LIN {X 0,Y 340.799,Z 465.238,A -85,B 0,C 180,E1 -14193.019,E2 -14193.019} C_VEL
LIN {X 0,Y 340.748,Z 465.291,A -85,B 0,C 180,E1 -14195.638,E2 -14195.638} C_VEL
LIN {X 0,Y 340.726,Z 465.225,A -85,B 0,C 180,E1 -14199.473,E2 -14199.473} C_VEL
LIN {X 0,Y 340.851,Z 465.236,A -85,B 0,C 180,E1 -14201.984,E2 -14201.984} C_VEL
LIN {X 0,Y 340.863,Z 465.263,A -85,B 0,C 180,E1 -14205.705,E2 -14205.705} C_VEL
LIN {X 0,Y 340.864,Z 465.273,A -85,B 0,C 180,E1 -14209.306,E2 -14209.306} C_VEL
LIN {X 0,Y 341.054,Z 465.245,A -85,B 0,C 180,E1 -14212.898,E2 -14212.898} C_VEL
LIN {X 0,Y 341.162,Z 465.23,A -85,B 0,C 180,E1 -14217.638,E2 -14217.638} C_VEL
LIN {X 0,Y 341.269,Z 465.216,A -85,B 0,C 180,E1 -14220,E2 -14220} C_VEL
LIN {X 0,Y 341.163,Z 465.221,A -85,B 0,C 180,E1 -14222.361,E2 -14222.361} C_VEL
LIN {X 0,Y 341.054,Z 465.234,A -85,B 0,C 180,E1 -14227.102,E2 -14227.102} C_VEL
LIN {X 0,Y 340.863,Z 465.256,A -85,B 0,C 180,E1 -14230.694,E2 -14230.694} C_VEL
LIN {X 0,Y 340.856,Z 465.271,A -85,B 0,C 180,E1 -14234.325,E2 -14234.325} C_VEL
LIN {X 0,Y 340.83,Z 465.282,A -85,B 0,C 180,E1 -14238.466,E2 -14238.466} C_VEL
LIN {X 0,Y 340.713,Z 465.293,A -85,B 0,C 180,E1 -14241.843,E2 -14241.843} C_VEL
LIN {X 0,Y 340.764,Z 465.235,A -85,B 0,C 180,E1 -14245.665,E2 -14245.665} C_VEL
LIN {X 0,Y 340.735,Z 465.25,A -85,B 0,C 180,E1 -14248.32,E2 -14248.32} C_VEL
LIN {X 0,Y 340.697,Z 465.294,A -85,B 0,C 180,E1 -14251.044,E2 -14251.044} C_VEL
LIN {X 0,Y 340.712,Z 465.253,A -85,B 0,C 180,E1 -14255.279,E2 -14255.279} C_VEL
LIN {X 0,Y 340.719,Z 465.295,A -85,B 0,C 180,E1 -14258.39,E2 -14258.39} C_VEL
LIN {X 0,Y 340.719,Z 465.295,A -85,B 0,C 180,E1 -14261.304,E2 -14261.304} C_VEL
LIN {X 0,Y 340.717,Z 465.295,A -85,B 0,C 180,E1 -14264.532,E2 -14264.532} C_VEL
LIN {X 0,Y 340.728,Z 465.294,A -85,B 0,C 180,E1 -14267.948,E2 -14267.948} C_VEL
LIN {X 0,Y 340.723,Z 465.445,A -85,B 0,C 180,E1 -14269.848,E2 -14269.848} C_VEL
LIN {X 0,Y 341.012,Z 466.611,A -85,B 0,C 180,E1 -14270.401,E2 -14270.401} C_VEL
LIN {X 0,Y 342.25,Z 468.887,A -85,B 0,C 180,E1 -14271.014,E2 -14271.014} C_VEL
LIN {X 0,Y 344.629,Z 470.782,A -85,B 0,C 180,E1 -14272.06,E2 -14272.06} C_VEL
LIN {X 0,Y 345.88,Z 471.693,A -85,B 0,C 180,E1 -14272.605,E2 -14272.605} C_VEL
LIN {X 0,Y 347.625,Z 474.655,A -85,B 0,C 180,E1 -14273.477,E2 -14273.477} C_VEL
LIN {X 0,Y 350.309,Z 476.774,A -85,B 0,C 180,E1 -14274.708,E2 -14274.708} C_VEL
LIN {X 0,Y 351.421,Z 477.644,A -85,B 0,C 180,E1 -14275.211,E2 -14275.211} C_VEL
LIN {X 0,Y 353.186,Z 480.48,A -85,B 0,C 180,E1 -14276.141,E2 -14276.141} C_VEL
LIN {X 0,Y 355.66,Z 482.592,A -85,B 0,C 180,E1 -14277.346,E2 -14277.346} C_VEL
LIN {X 0,Y 357.075,Z 483.51,A -85,B 0,C 180,E1 -14278.024,E2 -14278.024} C_VEL
LIN {X 0,Y 359.092,Z 486.493,A -85,B 0,C 180,E1 -14279.137,E2 -14279.137} C_VEL
LIN {X 0,Y 361.635,Z 488.623,A -85,B 0,C 180,E1 -14280.474,E2 -14280.474} C_VEL
LIN {X 0,Y 363.122,Z 489.584,A -85,B 0,C 180,E1 -14281.247,E2 -14281.247} C_VEL
LIN {X 0,Y 365.429,Z 492.822,A -85,B 0,C 180,E1 -14282.618,E2 -14282.618} C_VEL
LIN {X 0,Y 368.413,Z 495.129,A -85,B 0,C 180,E1 -14284.366,E2 -14284.366} C_VEL
LIN {X 0,Y 369.281,Z 495.706,A -85,B 0,C 180,E1 -14284.883,E2 -14284.883} C_VEL
LIN {X 0,Y 371.456,Z 498.808,A -85,B 0,C 180,E1 -14286.343,E2 -14286.343} C_VEL
LIN {X 0,Y 373.823,Z 500.83,A -85,B 0,C 180,E1 -14287.914,E2 -14287.914} C_VEL
LIN {X 0,Y 375.91,Z 502.055,A -85,B 0,C 180,E1 -14289.347,E2 -14289.347} C_VEL
LIN {X 0,Y 377.976,Z 505.06,A -85,B 0,C 180,E1 -14291.017,E2 -14291.017} C_VEL
LIN {X 0,Y 380.522,Z 507.196,A -85,B 0,C 180,E1 -14293.159,E2 -14293.159} C_VEL
LIN {X 0,Y 382.957,Z 508.62,A -85,B 0,C 180,E1 -14295.383,E2 -14295.383} C_VEL
LIN {X 0,Y 384.39,Z 510.97,A -85,B 0,C 180,E1 -14297.071,E2 -14297.071} C_VEL
LIN {X 0,Y 386.194,Z 512.79,A -85,B 0,C 180,E1 -14299.323,E2 -14299.323} C_VEL
LIN {X 0,Y 387.761,Z 513.727,A -85,B 0,C 180,E1 -14301.663,E2 -14301.663} C_VEL
LIN {X 0,Y 389.276,Z 514.525,A -85,B 0,C 180,E1 -14304.821,E2 -14304.821} C_VEL
LIN {X 0,Y 389.886,Z 514.854,A -85,B 0,C 180,E1 -14306.9,E2 -14306.9} C_VEL
LIN {X 0,Y 390.177,Z 515.105,A -85,B 0,C 180,E1 -14308.968,E2 -14308.968} C_VEL
LIN {X 0,Y 390.177,Z 515.108,A -85,B 0,C 180,E1 -14311.032,E2 -14311.032} C_VEL
LIN {X 0,Y 389.886,Z 514.854,A -85,B 0,C 180,E1 -14313.1,E2 -14313.1} C_VEL
LIN {X 0,Y 389.276,Z 514.517,A -85,B 0,C 180,E1 -14315.179,E2 -14315.179} C_VEL
LIN {X 0,Y 388.018,Z 513.851,A -85,B 0,C 180,E1 -14317.882,E2 -14317.882} C_VEL
LIN {X 0,Y 386.325,Z 512.888,A -85,B 0,C 180,E1 -14320.481,E2 -14320.481} C_VEL
LIN {X 0,Y 384.529,Z 511.148,A -85,B 0,C 180,E1 -14322.765,E2 -14322.765} C_VEL
LIN {X 0,Y 383.033,Z 508.786,A -85,B 0,C 180,E1 -14324.521,E2 -14324.521} C_VEL
LIN {X 0,Y 381.452,Z 507.625,A -85,B 0,C 180,E1 -14326.043,E2 -14326.043} C_VEL
LIN {X 0,Y 378.941,Z 506.028,A -85,B 0,C 180,E1 -14328.17,E2 -14328.17} C_VEL
LIN {X 0,Y 376.883,Z 503.704,A -85,B 0,C 180,E1 -14329.842,E2 -14329.842} C_VEL
LIN {X 0,Y 375.682,Z 501.75,A -85,B 0,C 180,E1 -14330.82,E2 -14330.82} C_VEL
LIN {X 0,Y 372.73,Z 500.116,A -85,B 0,C 180,E1 -14332.801,E2 -14332.801} C_VEL
LIN {X 0,Y 370.289,Z 497.364,A -85,B 0,C 180,E1 -14334.444,E2 -14334.444} C_VEL
LIN {X 0,Y 368.921,Z 495.376,A -85,B 0,C 180,E1 -14335.338,E2 -14335.338} C_VEL
LIN {X 0,Y 365.831,Z 493.26,A -85,B 0,C 180,E1 -14337.137,E2 -14337.137} C_VEL
LIN {X 0,Y 363.334,Z 489.978,A -85,B 0,C 180,E1 -14338.618,E2 -14338.618} C_VEL
LIN {X 0,Y 362.471,Z 489.035,A -85,B 0,C 180,E1 -14339.107,E2 -14339.107} C_VEL
LIN {X 0,Y 359.635,Z 487.068,A -85,B 0,C 180,E1 -14340.582,E2 -14340.582} C_VEL
LIN {X 0,Y 357.4,Z 484.129,A -85,B 0,C 180,E1 -14341.799,E2 -14341.799} C_VEL
LIN {X 0,Y 356.762,Z 483.15,A -85,B 0,C 180,E1 -14342.132,E2 -14342.132} C_VEL
LIN {X 0,Y 353.946,Z 481.231,A -85,B 0,C 180,E1 -14343.494,E2 -14343.494} C_VEL
LIN {X 0,Y 351.935,Z 478.654,A -85,B 0,C 180,E1 -14344.511,E2 -14344.511} C_VEL
LIN {X 0,Y 351.246,Z 477.269,A -85,B 0,C 180,E1 -14344.88,E2 -14344.88} C_VEL
LIN {X 0,Y 348.17,Z 475.197,A -85,B 0,C 180,E1 -14346.279,E2 -14346.279} C_VEL
LIN {X 0,Y 346.328,Z 472.631,A -85,B 0,C 180,E1 -14347.157,E2 -14347.157} C_VEL
LIN {X 0,Y 345.416,Z 471.159,A -85,B 0,C 180,E1 -14347.617,E2 -14347.617} C_VEL
LIN {X 0,Y 342.655,Z 469.35,A -85,B 0,C 180,E1 -14348.796,E2 -14348.796} C_VEL
LIN {X 0,Y 341.302,Z 467.35,A -85,B 0,C 180,E1 -14349.427,E2 -14349.427} C_VEL
LIN {X 0,Y 340.805,Z 465.884,A -85,B 0,C 180,E1 -14349.863,E2 -14349.863} C_VEL
LIN {X 0,Y 340.725,Z 465.368,A -85,B 0,C 180,E1 -14350.255,E2 -14350.255} C_VEL
LIN {X 0,Y 340.701,Z 465.298,A -85,B 0,C 180,E1 -14353.782,E2 -14353.782} C_VEL
LIN {X 0,Y 340.734,Z 465.294,A -85,B 0,C 180,E1 -14357.105,E2 -14357.105} C_VEL
LIN {X 0,Y 340.73,Z 465.294,A -85,B 0,C 180,E1 -14360.252,E2 -14360.252} C_VEL
LIN {X 0,Y 340.706,Z 465.281,A -85,B 0,C 180,E1 -14363.558,E2 -14363.558} C_VEL
LIN {X 0,Y 340.685,Z 465.246,A -85,B 0,C 180,E1 -14366.153,E2 -14366.153} C_VEL
LIN {X 0,Y 340.768,Z 465.28,A -85,B 0,C 180,E1 -14370.332,E2 -14370.332} C_VEL
LIN {X 0,Y 340.797,Z 465.225,A -85,B 0,C 180,E1 -14373.02,E2 -14373.02} C_VEL
LIN {X 0,Y 340.752,Z 465.241,A -85,B 0,C 180,E1 -14374.696,E2 -14374.696} C_VEL
LIN {X 0,Y 340.069,Z 465.349,A -85,B 0,C 180,E1 -14375.682,E2 -14375.682} C_VEL
LIN {X 0,Y 337.172,Z 465.738,A -85,B 0,C 180,E1 -14377.286,E2 -14377.286} C_VEL
LIN {X 0,Y 334.749,Z 466.031,A -85,B 0,C 180,E1 -14378.585,E2 -14378.585} C_VEL
LIN {X 0,Y 333.75,Z 466.146,A -85,B 0,C 180,E1 -14379.592,E2 -14379.592} C_VEL
LIN {X 0,Y 333.69,Z 466.154,A -85,B 0,C 180,E1 -14379.932,E2 -14379.932} C_VEL
LIN {X 0,Y 333.738,Z 466.154,A -85,B 0,C 180,E1 -14382.854,E2 -14382.854} C_VEL
LIN {X 0,Y 333.789,Z 466.155,A -85,B 0,C 180,E1 -14386.609,E2 -14386.609} C_VEL
LIN {X 0,Y 333.853,Z 466.142,A -85,B 0,C 180,E1 -14390.305,E2 -14390.305} C_VEL
LIN {X 0,Y 334.006,Z 466.114,A -85,B 0,C 180,E1 -14392.747,E2 -14392.747} C_VEL
LIN {X 0,Y 333.805,Z 466.147,A -85,B 0,C 180,E1 -14395.169,E2 -14395.169} C_VEL
LIN {X 0,Y 334.1,Z 466.103,A -85,B 0,C 180,E1 -14397.589,E2 -14397.589} C_VEL
LIN {X 0,Y 334.221,Z 466.094,A -85,B 0,C 180,E1 -14400,E2 -14400} C_VEL
LIN {X 0,Y 334.099,Z 466.109,A -85,B 0,C 180,E1 -14402.411,E2 -14402.411} C_VEL
LIN {X 0,Y 334.01,Z 466.129,A -85,B 0,C 180,E1 -14406.039,E2 -14406.039} C_VEL
LIN {X 0,Y 333.952,Z 466.115,A -85,B 0,C 180,E1 -14408.472,E2 -14408.472} C_VEL
LIN {X 0,Y 333.784,Z 466.146,A -85,B 0,C 180,E1 -14412.155,E2 -14412.155} C_VEL
LIN {X 0,Y 333.771,Z 466.158,A -85,B 0,C 180,E1 -14415.887,E2 -14415.887} C_VEL
LIN {X 0,Y 333.789,Z 466.1,A -85,B 0,C 180,E1 -14418.655,E2 -14418.655} C_VEL
LIN {X 0,Y 333.65,Z 466.134,A -85,B 0,C 180,E1 -14422.281,E2 -14422.281} C_VEL
LIN {X 0,Y 333.73,Z 466.133,A -85,B 0,C 180,E1 -14426.247,E2 -14426.247} C_VEL
LIN {X 0,Y 333.706,Z 466.111,A -85,B 0,C 180,E1 -14428.973,E2 -14428.973} C_VEL
LIN {X 0,Y 333.646,Z 466.172,A -85,B 0,C 180,E1 -14432.59,E2 -14432.59} C_VEL
LIN {X 0,Y 333.672,Z 466.144,A -85,B 0,C 180,E1 -14436.139,E2 -14436.139} C_VEL
LIN {X 0,Y 333.678,Z 466.146,A -85,B 0,C 180,E1 -14439.188,E2 -14439.188} C_VEL
LIN {X 0,Y 333.708,Z 466.29,A -85,B 0,C 180,E1 -14441.258,E2 -14441.258} C_VEL
LIN {X 0,Y 336.781,Z 476.03,A -85,B 0,C 180,E1 -14444.671,E2 -14444.671} C_VEL
LIN {X 0,Y 337.849,Z 478.396,A -85,B 0,C 180,E1 -14445.014,E2 -14445.014} C_VEL
LIN {X 0,Y 341.276,Z 483.882,A -85,B 0,C 180,E1 -14445.739,E2 -14445.739} C_VEL
LIN {X 0,Y 349.072,Z 497.083,A -85,B 0,C 180,E1 -14447.326,E2 -14447.326} C_VEL
LIN {X 0,Y 358.673,Z 515.254,A -85,B 0,C 180,E1 -14449.186,E2 -14449.186} C_VEL
LIN {X 0,Y 366.818,Z 532.432,A -85,B 0,C 180,E1 -14450.694,E2 -14450.694} C_VEL
LIN {X 0,Y 368.049,Z 538.307,A -85,B 0,C 180,E1 -14450.994,E2 -14450.994} C_VEL
LIN {X 0,Y 363.639,Z 661.533,A -85,B 0,C 180,E1 -14453.452,E2 -14453.452} C_VEL
LIN {X 0,Y 362.413,Z 691.653,A -85,B 0,C 180,E1 -14454.084,E2 -14454.084} C_VEL
LIN {X 0,Y 361.365,Z 705.109,A -85,B 0,C 180,E1 -14454.479,E2 -14454.479} C_VEL
LIN {X 0,Y 359.961,Z 718.486,A -85,B 0,C 180,E1 -14455.005,E2 -14455.005} C_VEL
LIN {X 0,Y 358.069,Z 734.159,A -85,B 0,C 180,E1 -14455.818,E2 -14455.818} C_VEL
LIN {X 0,Y 355.544,Z 750.452,A -85,B 0,C 180,E1 -14456.904,E2 -14456.904} C_VEL
LIN {X 0,Y 353.23,Z 763.836,A -85,B 0,C 180,E1 -14458.013,E2 -14458.013} C_VEL
LIN {X 0,Y 350.74,Z 776.671,A -85,B 0,C 180,E1 -14459.274,E2 -14459.274} C_VEL
LIN {X 0,Y 348.622,Z 786.926,A -85,B 0,C 180,E1 -14460.442,E2 -14460.442} C_VEL
LIN {X 0,Y 346.254,Z 797.637,A -85,B 0,C 180,E1 -14461.842,E2 -14461.842} C_VEL
LIN {X 0,Y 344.049,Z 807.328,A -85,B 0,C 180,E1 -14463.295,E2 -14463.295} C_VEL
LIN {X 0,Y 342.031,Z 816.281,A -85,B 0,C 180,E1 -14464.827,E2 -14464.827} C_VEL
LIN {X 0,Y 339.631,Z 826.499,A -85,B 0,C 180,E1 -14466.849,E2 -14466.849} C_VEL
LIN {X 0,Y 337.855,Z 834.392,A -85,B 0,C 180,E1 -14468.653,E2 -14468.653} C_VEL
LIN {X 0,Y 336.381,Z 841.359,A -85,B 0,C 180,E1 -14470.471,E2 -14470.471} C_VEL
LIN {X 0,Y 335.184,Z 847.502,A -85,B 0,C 180,E1 -14472.301,E2 -14472.301} C_VEL
LIN {X 0,Y 333.91,Z 854.451,A -85,B 0,C 180,E1 -14474.747,E2 -14474.747} C_VEL
LIN {X 0,Y 332.975,Z 860.207,A -85,B 0,C 180,E1 -14477.196,E2 -14477.196} C_VEL
LIN {X 0,Y 332.45,Z 863.818,A -85,B 0,C 180,E1 -14479.032,E2 -14479.032} C_VEL
LIN {X 0,Y 332.118,Z 867.67,A -85,B 0,C 180,E1 -14481.482,E2 -14481.482} C_VEL
LIN {X 0,Y 332.029,Z 870.521,A -85,B 0,C 180,E1 -14483.925,E2 -14483.925} C_VEL
LIN {X 0,Y 331.964,Z 872.403,A -85,B 0,C 180,E1 -14486.359,E2 -14486.359} C_VEL
LIN {X 0,Y 331.902,Z 873.076,A -85,B 0,C 180,E1 -14487.573,E2 -14487.573} C_VEL
LIN {X 0,Y 331.911,Z 873.548,A -85,B 0,C 180,E1 -14490,E2 -14490} C_VEL
LIN {X 0,Y 331.902,Z 873.076,A -85,B 0,C 180,E1 -14492.427,E2 -14492.427} C_VEL
LIN {X 0,Y 331.936,Z 871.654,A -85,B 0,C 180,E1 -14494.858,E2 -14494.858} C_VEL
LIN {X 0,Y 332.033,Z 869.271,A -85,B 0,C 180,E1 -14497.296,E2 -14497.296} C_VEL
LIN {X 0,Y 332.347,Z 864.858,A -85,B 0,C 180,E1 -14500.355,E2 -14500.355} C_VEL
LIN {X 0,Y 332.783,Z 861.493,A -85,B 0,C 180,E1 -14502.192,E2 -14502.192} C_VEL
LIN {X 0,Y 333.616,Z 855.994,A -85,B 0,C 180,E1 -14504.643,E2 -14504.643} C_VEL
LIN {X 0,Y 334.458,Z 851.135,A -85,B 0,C 180,E1 -14506.479,E2 -14506.479} C_VEL
LIN {X 0,Y 335.999,Z 843.467,A -85,B 0,C 180,E1 -14508.917,E2 -14508.917} C_VEL
LIN {X 0,Y 337.306,Z 836.81,A -85,B 0,C 180,E1 -14510.744,E2 -14510.744} C_VEL
LIN {X 0,Y 339.006,Z 829.257,A -85,B 0,C 180,E1 -14512.552,E2 -14512.552} C_VEL
LIN {X 0,Y 341.098,Z 820.675,A -85,B 0,C 180,E1 -14514.335,E2 -14514.335} C_VEL
LIN {X 0,Y 343.221,Z 810.88,A -85,B 0,C 180,E1 -14516.119,E2 -14516.119} C_VEL
LIN {X 0,Y 345.731,Z 799.648,A -85,B 0,C 180,E1 -14517.874,E2 -14517.874} C_VEL
LIN {X 0,Y 348.088,Z 789.167,A -85,B 0,C 180,E1 -14519.282,E2 -14519.282} C_VEL
LIN {X 0,Y 350.131,Z 779.54,A -85,B 0,C 180,E1 -14520.419,E2 -14520.419} C_VEL
LIN {X 0,Y 352.331,Z 768.335,A -85,B 0,C 180,E1 -14521.574,E2 -14521.574} C_VEL
LIN {X 0,Y 354.632,Z 755.677,A -85,B 0,C 180,E1 -14522.685,E2 -14522.685} C_VEL
LIN {X 0,Y 356.641,Z 743.661,A -85,B 0,C 180,E1 -14523.572,E2 -14523.572} C_VEL
LIN {X 0,Y 358.505,Z 730.453,A -85,B 0,C 180,E1 -14524.39,E2 -14524.39} C_VEL
LIN {X 0,Y 360.135,Z 717.326,A -85,B 0,C 180,E1 -14525.04,E2 -14525.04} C_VEL
LIN {X 0,Y 361.468,Z 704.407,A -85,B 0,C 180,E1 -14525.54,E2 -14525.54} C_VEL
LIN {X 0,Y 362.415,Z 691.653,A -85,B 0,C 180,E1 -14525.916,E2 -14525.916} C_VEL
LIN {X 0,Y 363.878,Z 654.368,A -85,B 0,C 180,E1 -14526.692,E2 -14526.692} C_VEL
LIN {X 0,Y 367.077,Z 565.249,A -85,B 0,C 180,E1 -14528.468,E2 -14528.468} C_VEL
LIN {X 0,Y 368.055,Z 538.146,A -85,B 0,C 180,E1 -14529.01,E2 -14529.01} C_VEL
LIN {X 0,Y 366.541,Z 531.775,A -85,B 0,C 180,E1 -14529.358,E2 -14529.358} C_VEL
LIN {X 0,Y 357.488,Z 512.916,A -85,B 0,C 180,E1 -14531.038,E2 -14531.038} C_VEL
LIN {X 0,Y 348.525,Z 496.099,A -85,B 0,C 180,E1 -14532.783,E2 -14532.783} C_VEL
LIN {X 0,Y 339.359,Z 480.633,A -85,B 0,C 180,E1 -14534.669,E2 -14534.669} C_VEL
LIN {X 0,Y 336.838,Z 476.211,A -85,B 0,C 180,E1 -14535.284,E2 -14535.284} C_VEL
LIN {X 0,Y 333.701,Z 466.326,A -85,B 0,C 180,E1 -14538.741,E2 -14538.741} C_VEL
LIN {X 0,Y 333.651,Z 466.176,A -85,B 0,C 180,E1 -14542.349,E2 -14542.349} C_VEL
LIN {X 0,Y 333.669,Z 466.135,A -85,B 0,C 180,E1 -14545.341,E2 -14545.341} C_VEL
LIN {X 0,Y 333.639,Z 466.176,A -85,B 0,C 180,E1 -14548.223,E2 -14548.223} C_VEL
LIN {X 0,Y 333.706,Z 466.111,A -85,B 0,C 180,E1 -14551.027,E2 -14551.027} C_VEL
LIN {X 0,Y 333.73,Z 466.132,A -85,B 0,C 180,E1 -14553.753,E2 -14553.753} C_VEL
LIN {X 0,Y 333.65,Z 466.134,A -85,B 0,C 180,E1 -14557.719,E2 -14557.719} C_VEL
LIN {X 0,Y 333.787,Z 466.104,A -85,B 0,C 180,E1 -14561.589,E2 -14561.589} C_VEL
LIN {X 0,Y 333.802,Z 466.143,A -85,B 0,C 180,E1 -14565.576,E2 -14565.576} C_VEL
LIN {X 0,Y 333.827,Z 466.15,A -85,B 0,C 180,E1 -14569.078,E2 -14569.078} C_VEL
LIN {X 0,Y 334.001,Z 466.121,A -85,B 0,C 180,E1 -14572.747,E2 -14572.747} C_VEL
LIN {X 0,Y 333.805,Z 466.146,A -85,B 0,C 180,E1 -14575.169,E2 -14575.169} C_VEL
LIN {X 0,Y 334.1,Z 466.108,A -85,B 0,C 180,E1 -14577.589,E2 -14577.589} C_VEL
LIN {X 0,Y 334.221,Z 466.093,A -85,B 0,C 180,E1 -14580,E2 -14580} C_VEL
LIN {X 0,Y 334.1,Z 466.1,A -85,B 0,C 180,E1 -14582.411,E2 -14582.411} C_VEL
LIN {X 0,Y 333.989,Z 466.11,A -85,B 0,C 180,E1 -14586.616,E2 -14586.616} C_VEL
LIN {X 0,Y 333.853,Z 466.141,A -85,B 0,C 180,E1 -14589.695,E2 -14589.695} C_VEL
LIN {X 0,Y 333.789,Z 466.155,A -85,B 0,C 180,E1 -14593.391,E2 -14593.391} C_VEL
LIN {X 0,Y 333.738,Z 466.154,A -85,B 0,C 180,E1 -14597.146,E2 -14597.146} C_VEL
LIN {X 0,Y 333.725,Z 466.152,A -85,B 0,C 180,E1 -14599.691,E2 -14599.691} C_VEL
LIN {X 0,Y 333.664,Z 466.164,A -85,B 0,C 180,E1 -14603.59,E2 -14603.59} C_VEL
LIN {X 0,Y 333.728,Z 466.104,A -85,B 0,C 180,E1 -14606.246,E2 -14606.246} C_VEL
LIN {X 0,Y 333.704,Z 466.14,A -85,B 0,C 180,E1 -14608.972,E2 -14608.972} C_VEL
LIN {X 0,Y 333.636,Z 466.136,A -85,B 0,C 180,E1 -14612.587,E2 -14612.587} C_VEL
LIN {X 0,Y 333.671,Z 466.147,A -85,B 0,C 180,E1 -14616.139,E2 -14616.139} C_VEL
LIN {X 0,Y 333.681,Z 466.173,A -85,B 0,C 180,E1 -14619.187,E2 -14619.187} C_VEL
LIN {X 0,Y 333.683,Z 466.171,A -85,B 0,C 180,E1 -14622.511,E2 -14622.511} C_VEL
LIN {X 0,Y 333.653,Z 466.174,A -85,B 0,C 180,E1 -14625.966,E2 -14625.966} C_VEL
LIN {X 0,Y 333.716,Z 466.35,A -85,B 0,C 180,E1 -14627.284,E2 -14627.284} C_VEL
LIN {X 0,Y 334.001,Z 467.585,A -85,B 0,C 180,E1 -14627.8,E2 -14627.8} C_VEL
LIN {X 0,Y 335.396,Z 469.981,A -85,B 0,C 180,E1 -14628.466,E2 -14628.466} C_VEL
LIN {X 0,Y 337.884,Z 471.863,A -85,B 0,C 180,E1 -14629.485,E2 -14629.485} C_VEL
LIN {X 0,Y 338.798,Z 472.664,A -85,B 0,C 180,E1 -14629.887,E2 -14629.887} C_VEL
LIN {X 0,Y 340.366,Z 475.312,A -85,B 0,C 180,E1 -14630.625,E2 -14630.625} C_VEL
LIN {X 0,Y 342.872,Z 477.456,A -85,B 0,C 180,E1 -14631.722,E2 -14631.722} C_VEL
LIN {X 0,Y 344.061,Z 478.298,A -85,B 0,C 180,E1 -14632.229,E2 -14632.229} C_VEL
LIN {X 0,Y 346.074,Z 481.409,A -85,B 0,C 180,E1 -14633.214,E2 -14633.214} C_VEL
LIN {X 0,Y 348.838,Z 483.58,A -85,B 0,C 180,E1 -14634.467,E2 -14634.467} C_VEL
LIN {X 0,Y 349.69,Z 484.296,A -85,B 0,C 180,E1 -14634.863,E2 -14634.863} C_VEL
LIN {X 0,Y 351.781,Z 487.31,A -85,B 0,C 180,E1 -14635.92,E2 -14635.92} C_VEL
LIN {X 0,Y 354.617,Z 489.628,A -85,B 0,C 180,E1 -14637.289,E2 -14637.289} C_VEL
LIN {X 0,Y 355.598,Z 490.455,A -85,B 0,C 180,E1 -14637.775,E2 -14637.775} C_VEL
LIN {X 0,Y 358.077,Z 493.716,A -85,B 0,C 180,E1 -14639.102,E2 -14639.102} C_VEL
LIN {X 0,Y 360.763,Z 495.744,A -85,B 0,C 180,E1 -14640.497,E2 -14640.497} C_VEL
LIN {X 0,Y 361.761,Z 496.461,A -85,B 0,C 180,E1 -14641.011,E2 -14641.011} C_VEL
LIN {X 0,Y 364.25,Z 499.79,A -85,B 0,C 180,E1 -14642.469,E2 -14642.469} C_VEL
LIN {X 0,Y 367.384,Z 502.135,A -85,B 0,C 180,E1 -14644.289,E2 -14644.289} C_VEL
LIN {X 0,Y 368.211,Z 502.958,A -85,B 0,C 180,E1 -14644.805,E2 -14644.805} C_VEL
LIN {X 0,Y 370.641,Z 506.172,A -85,B 0,C 180,E1 -14646.411,E2 -14646.411} C_VEL
LIN {X 0,Y 373.648,Z 508.333,A -85,B 0,C 180,E1 -14648.402,E2 -14648.402} C_VEL
LIN {X 0,Y 374.774,Z 509.041,A -85,B 0,C 180,E1 -14649.188,E2 -14649.188} C_VEL
LIN {X 0,Y 376.863,Z 511.983,A -85,B 0,C 180,E1 -14650.848,E2 -14650.848} C_VEL
LIN {X 0,Y 379.588,Z 514.233,A -85,B 0,C 180,E1 -14653.116,E2 -14653.116} C_VEL
LIN {X 0,Y 381.909,Z 515.568,A -85,B 0,C 180,E1 -14655.207,E2 -14655.207} C_VEL
LIN {X 0,Y 383.479,Z 518.067,A -85,B 0,C 180,E1 -14657.039,E2 -14657.039} C_VEL
LIN {X 0,Y 385.431,Z 519.973,A -85,B 0,C 180,E1 -14659.494,E2 -14659.494} C_VEL
LIN {X 0,Y 387.14,Z 520.894,A -85,B 0,C 180,E1 -14662.101,E2 -14662.101} C_VEL
LIN {X 0,Y 388.408,Z 521.561,A -85,B 0,C 180,E1 -14664.809,E2 -14664.809} C_VEL
LIN {X 0,Y 389.019,Z 521.9,A -85,B 0,C 180,E1 -14666.893,E2 -14666.893} C_VEL
LIN {X 0,Y 389.312,Z 522.151,A -85,B 0,C 180,E1 -14668.966,E2 -14668.966} C_VEL
LIN {X 0,Y 389.312,Z 522.154,A -85,B 0,C 180,E1 -14671.034,E2 -14671.034} C_VEL
LIN {X 0,Y 389.019,Z 521.9,A -85,B 0,C 180,E1 -14673.107,E2 -14673.107} C_VEL
LIN {X 0,Y 388.31,Z 521.48,A -85,B 0,C 180,E1 -14675.48,E2 -14675.48} C_VEL
LIN {X 0,Y 386.879,Z 520.77,A -85,B 0,C 180,E1 -14678.356,E2 -14678.356} C_VEL
LIN {X 0,Y 385.035,Z 519.643,A -85,B 0,C 180,E1 -14681.047,E2 -14681.047} C_VEL
LIN {X 0,Y 383.292,Z 517.821,A -85,B 0,C 180,E1 -14683.19,E2 -14683.19} C_VEL
LIN {X 0,Y 381.547,Z 515.224,A -85,B 0,C 180,E1 -14685.156,E2 -14685.156} C_VEL
LIN {X 0,Y 378.664,Z 513.605,A -85,B 0,C 180,E1 -14687.681,E2 -14687.681} C_VEL
LIN {X 0,Y 376.317,Z 511.354,A -85,B 0,C 180,E1 -14689.572,E2 -14689.572} C_VEL
LIN {X 0,Y 374.469,Z 508.696,A -85,B 0,C 180,E1 -14691.032,E2 -14691.032} C_VEL
LIN {X 0,Y 371.535,Z 506.981,A -85,B 0,C 180,E1 -14693.005,E2 -14693.005} C_VEL
LIN {X 0,Y 368.963,Z 504.114,A -85,B 0,C 180,E1 -14694.717,E2 -14694.717} C_VEL
LIN {X 0,Y 367.639,Z 502.248,A -85,B 0,C 180,E1 -14695.563,E2 -14695.563} C_VEL
LIN {X 0,Y 364.568,Z 500.105,A -85,B 0,C 180,E1 -14697.345,E2 -14697.345} C_VEL
LIN {X 0,Y 361.995,Z 496.856,A -85,B 0,C 180,E1 -14698.851,E2 -14698.851} C_VEL
LIN {X 0,Y 361.33,Z 496.008,A -85,B 0,C 180,E1 -14699.218,E2 -14699.218} C_VEL
LIN {X 0,Y 358.483,Z 494.098,A -85,B 0,C 180,E1 -14700.689,E2 -14700.689} C_VEL
LIN {X 0,Y 355.928,Z 490.993,A -85,B 0,C 180,E1 -14702.049,E2 -14702.049} C_VEL
LIN {X 0,Y 355.336,Z 489.998,A -85,B 0,C 180,E1 -14702.366,E2 -14702.366} C_VEL
LIN {X 0,Y 352.412,Z 487.954,A -85,B 0,C 180,E1 -14703.77,E2 -14703.77} C_VEL
LIN {X 0,Y 350.116,Z 485.046,A -85,B 0,C 180,E1 -14704.922,E2 -14704.922} C_VEL
LIN {X 0,Y 349.317,Z 483.857,A -85,B 0,C 180,E1 -14705.316,E2 -14705.316} C_VEL
LIN {X 0,Y 346.252,Z 481.607,A -85,B 0,C 180,E1 -14706.704,E2 -14706.704} C_VEL
LIN {X 0,Y 344.287,Z 478.716,A -85,B 0,C 180,E1 -14707.664,E2 -14707.664} C_VEL
LIN {X 0,Y 343.675,Z 477.863,A -85,B 0,C 180,E1 -14707.943,E2 -14707.943} C_VEL
LIN {X 0,Y 340.917,Z 475.912,A -85,B 0,C 180,E1 -14709.138,E2 -14709.138} C_VEL
LIN {X 0,Y 339.142,Z 473.436,A -85,B 0,C 180,E1 -14709.938,E2 -14709.938} C_VEL
LIN {X 0,Y 338.385,Z 472.108,A -85,B 0,C 180,E1 -14710.305,E2 -14710.305} C_VEL
LIN {X 0,Y 335.698,Z 470.334,A -85,B 0,C 180,E1 -14711.401,E2 -14711.401} C_VEL
LIN {X 0,Y 334.143,Z 467.942,A -85,B 0,C 180,E1 -14712.123,E2 -14712.123} C_VEL
LIN {X 0,Y 333.767,Z 466.637,A -85,B 0,C 180,E1 -14712.526,E2 -14712.526} C_VEL
LIN {X 0,Y 333.668,Z 466.18,A -85,B 0,C 180,E1 -14713.215,E2 -14713.215} C_VEL
LIN {X 0,Y 333.663,Z 466.174,A -85,B 0,C 180,E1 -14715.967,E2 -14715.967} C_VEL
LIN {X 0,Y 333.695,Z 466.17,A -85,B 0,C 180,E1 -14719.304,E2 -14719.304} C_VEL
LIN {X 0,Y 333.662,Z 466.169,A -85,B 0,C 180,E1 -14723.167,E2 -14723.167} C_VEL
LIN {X 0,Y 333.667,Z 466.122,A -85,B 0,C 180,E1 -14725.341,E2 -14725.341} C_VEL
LIN {X 0,Y 333.696,Z 466.169,A -85,B 0,C 180,E1 -14729.71,E2 -14729.71} C_VEL
LIN {X 0,Y 333.737,Z 466.108,A -85,B 0,C 180,E1 -14732.401,E2 -14732.401} C_VEL
LIN {X 0,Y 333.718,Z 466.124,A -85,B 0,C 180,E1 -14735.09,E2 -14735.09} C_VEL
LIN {X 0,Y 333.666,Z 466.158,A -85,B 0,C 180,E1 -14739.019,E2 -14739.019} C_VEL
LIN {X 0,Y 333.69,Z 466.154,A -85,B 0,C 180,E1 -14739.932,E2 -14739.932} C_VEL
LIN {X 0,Y 333.082,Z 466.24,A -85,B 0,C 180,E1 -14740.939,E2 -14740.939} C_VEL
LIN {X 0,Y 330.26,Z 466.592,A -85,B 0,C 180,E1 -14742.579,E2 -14742.579} C_VEL
LIN {X 0,Y 327.845,Z 466.883,A -85,B 0,C 180,E1 -14743.907,E2 -14743.907} C_VEL
LIN {X 0,Y 326.824,Z 467.008,A -85,B 0,C 180,E1 -14744.935,E2 -14744.935} C_VEL
LIN {X 0,Y 326.75,Z 467.021,A -85,B 0,C 180,E1 -14745.283,E2 -14745.283} C_VEL
LIN {X 0,Y 326.762,Z 467.011,A -85,B 0,C 180,E1 -14748.839,E2 -14748.839} C_VEL
LIN {X 0,Y 326.96,Z 466.993,A -85,B 0,C 180,E1 -14752.59,E2 -14752.59} C_VEL
LIN {X 0,Y 326.772,Z 467.022,A -85,B 0,C 180,E1 -14755.065,E2 -14755.065} C_VEL
LIN {X 0,Y 327.041,Z 466.982,A -85,B 0,C 180,E1 -14757.537,E2 -14757.537} C_VEL
LIN {X 0,Y 327.173,Z 466.972,A -85,B 0,C 180,E1 -14760,E2 -14760} C_VEL
LIN {X 0,Y 327.04,Z 466.987,A -85,B 0,C 180,E1 -14762.464,E2 -14762.464} C_VEL
LIN {X 0,Y 326.985,Z 467.003,A -85,B 0,C 180,E1 -14766.17,E2 -14766.17} C_VEL
LIN {X 0,Y 326.799,Z 467.016,A -85,B 0,C 180,E1 -14769.907,E2 -14769.907} C_VEL
LIN {X 0,Y 326.752,Z 467.014,A -85,B 0,C 180,E1 -14773.686,E2 -14773.686} C_VEL
LIN {X 0,Y 326.692,Z 467.01,A -85,B 0,C 180,E1 -14777.528,E2 -14777.528} C_VEL
LIN {X 0,Y 326.651,Z 466.974,A -85,B 0,C 180,E1 -14780.136,E2 -14780.136} C_VEL
LIN {X 0,Y 326.643,Z 467.048,A -85,B 0,C 180,E1 -14784.13,E2 -14784.13} C_VEL
LIN {X 0,Y 326.679,Z 466.995,A -85,B 0,C 180,E1 -14786.858,E2 -14786.858} C_VEL
LIN {X 0,Y 326.636,Z 467.02,A -85,B 0,C 180,E1 -14790.613,E2 -14790.613} C_VEL
LIN {X 0,Y 326.604,Z 467.019,A -85,B 0,C 180,E1 -14794.02,E2 -14794.02} C_VEL
LIN {X 0,Y 326.625,Z 467.045,A -85,B 0,C 180,E1 -14797.24,E2 -14797.24} C_VEL
LIN {X 0,Y 326.65,Z 467.151,A -85,B 0,C 180,E1 -14800.2,E2 -14800.2} C_VEL
LIN {X 0,Y 329.467,Z 475.897,A -85,B 0,C 180,E1 -14803.415,E2 -14803.415} C_VEL
LIN {X 0,Y 332.332,Z 480.715,A -85,B 0,C 180,E1 -14804.132,E2 -14804.132} C_VEL
LIN {X 0,Y 339.589,Z 492.764,A -85,B 0,C 180,E1 -14805.72,E2 -14805.72} C_VEL
LIN {X 0,Y 347.23,Z 506.263,A -85,B 0,C 180,E1 -14807.3,E2 -14807.3} C_VEL
LIN {X 0,Y 356.44,Z 524.382,A -85,B 0,C 180,E1 -14809.115,E2 -14809.115} C_VEL
LIN {X 0,Y 361.7,Z 535.896,A -85,B 0,C 180,E1 -14810.119,E2 -14810.119} C_VEL
LIN {X 0,Y 362.496,Z 539.647,A -85,B 0,C 180,E1 -14810.318,E2 -14810.318} C_VEL
LIN {X 0,Y 357.961,Z 661.323,A -85,B 0,C 180,E1 -14812.775,E2 -14812.775} C_VEL
LIN {X 0,Y 356.676,Z 691.443,A -85,B 0,C 180,E1 -14813.413,E2 -14813.413} C_VEL
LIN {X 0,Y 355.524,Z 705.9,A -85,B 0,C 180,E1 -14813.848,E2 -14813.848} C_VEL
LIN {X 0,Y 353.84,Z 721.343,A -85,B 0,C 180,E1 -14814.483,E2 -14814.483} C_VEL
LIN {X 0,Y 351.496,Z 738.469,A -85,B 0,C 180,E1 -14815.448,E2 -14815.448} C_VEL
LIN {X 0,Y 349.258,Z 751.982,A -85,B 0,C 180,E1 -14816.402,E2 -14816.402} C_VEL
LIN {X 0,Y 347.187,Z 763.625,A -85,B 0,C 180,E1 -14817.388,E2 -14817.388} C_VEL
LIN {X 0,Y 344.58,Z 776.454,A -85,B 0,C 180,E1 -14818.662,E2 -14818.662} C_VEL
LIN {X 0,Y 342.294,Z 787.09,A -85,B 0,C 180,E1 -14819.896,E2 -14819.896} C_VEL
LIN {X 0,Y 339.677,Z 798.43,A -85,B 0,C 180,E1 -14821.416,E2 -14821.416} C_VEL
LIN {X 0,Y 337.178,Z 808.891,A -85,B 0,C 180,E1 -14823.042,E2 -14823.042} C_VEL
LIN {X 0,Y 335.326,Z 816.805,A -85,B 0,C 180,E1 -14824.444,E2 -14824.444} C_VEL
LIN {X 0,Y 333.006,Z 826.285,A -85,B 0,C 180,E1 -14826.361,E2 -14826.361} C_VEL
LIN {X 0,Y 331.131,Z 834.179,A -85,B 0,C 180,E1 -14828.197,E2 -14828.197} C_VEL
LIN {X 0,Y 329.332,Z 842.198,A -85,B 0,C 180,E1 -14830.361,E2 -14830.361} C_VEL
LIN {X 0,Y 327.907,Z 849.105,A -85,B 0,C 180,E1 -14832.539,E2 -14832.539} C_VEL
LIN {X 0,Y 326.94,Z 854.237,A -85,B 0,C 180,E1 -14834.413,E2 -14834.413} C_VEL
LIN {X 0,Y 326.222,Z 858.709,A -85,B 0,C 180,E1 -14836.292,E2 -14836.292} C_VEL
LIN {X 0,Y 325.427,Z 863.607,A -85,B 0,C 180,E1 -14838.793,E2 -14838.793} C_VEL
LIN {X 0,Y 325.047,Z 867.458,A -85,B 0,C 180,E1 -14841.295,E2 -14841.295} C_VEL
LIN {X 0,Y 324.944,Z 870.311,A -85,B 0,C 180,E1 -14843.792,E2 -14843.792} C_VEL
LIN {X 0,Y 324.869,Z 872.193,A -85,B 0,C 180,E1 -14846.279,E2 -14846.279} C_VEL
LIN {X 0,Y 324.822,Z 872.867,A -85,B 0,C 180,E1 -14847.52,E2 -14847.52} C_VEL
LIN {X 0,Y 324.818,Z 873.339,A -85,B 0,C 180,E1 -14850,E2 -14850} C_VEL
LIN {X 0,Y 324.822,Z 872.867,A -85,B 0,C 180,E1 -14852.48,E2 -14852.48} C_VEL
LIN {X 0,Y 324.85,Z 871.444,A -85,B 0,C 180,E1 -14854.964,E2 -14854.964} C_VEL
LIN {X 0,Y 324.948,Z 869.06,A -85,B 0,C 180,E1 -14857.456,E2 -14857.456} C_VEL
LIN {X 0,Y 325.283,Z 864.646,A -85,B 0,C 180,E1 -14860.582,E2 -14860.582} C_VEL
LIN {X 0,Y 325.747,Z 861.28,A -85,B 0,C 180,E1 -14862.459,E2 -14862.459} C_VEL
LIN {X 0,Y 326.667,Z 855.782,A -85,B 0,C 180,E1 -14864.961,E2 -14864.961} C_VEL
LIN {X 0,Y 327.566,Z 850.922,A -85,B 0,C 180,E1 -14866.836,E2 -14866.836} C_VEL
LIN {X 0,Y 329.157,Z 843.253,A -85,B 0,C 180,E1 -14869.326,E2 -14869.326} C_VEL
LIN {X 0,Y 330.56,Z 836.597,A -85,B 0,C 180,E1 -14871.188,E2 -14871.188} C_VEL
LIN {X 0,Y 332.334,Z 829.043,A -85,B 0,C 180,E1 -14873.03,E2 -14873.03} C_VEL
LIN {X 0,Y 334.53,Z 820.462,A -85,B 0,C 180,E1 -14874.845,E2 -14874.845} C_VEL
LIN {X 0,Y 336.776,Z 810.667,A -85,B 0,C 180,E1 -14876.658,E2 -14876.658} C_VEL
LIN {X 0,Y 339.154,Z 800.442,A -85,B 0,C 180,E1 -14878.295,E2 -14878.295} C_VEL
LIN {X 0,Y 341.369,Z 791.02,A -85,B 0,C 180,E1 -14879.61,E2 -14879.61} C_VEL
LIN {X 0,Y 343.739,Z 780.369,A -85,B 0,C 180,E1 -14880.91,E2 -14880.91} C_VEL
LIN {X 0,Y 346.258,Z 768.124,A -85,B 0,C 180,E1 -14882.194,E2 -14882.194} C_VEL
LIN {X 0,Y 348.331,Z 757.207,A -85,B 0,C 180,E1 -14883.18,E2 -14883.18} C_VEL
LIN {X 0,Y 350.558,Z 744.476,A -85,B 0,C 180,E1 -14884.148,E2 -14884.148} C_VEL
LIN {X 0,Y 352.459,Z 731.588,A -85,B 0,C 180,E1 -14884.97,E2 -14884.97} C_VEL
LIN {X 0,Y 354.253,Z 717.807,A -85,B 0,C 180,E1 -14885.671,E2 -14885.671} C_VEL
LIN {X 0,Y 355.602,Z 705.296,A -85,B 0,C 180,E1 -14886.17,E2 -14886.17} C_VEL
LIN {X 0,Y 356.679,Z 691.443,A -85,B 0,C 180,E1 -14886.586,E2 -14886.586} C_VEL
LIN {X 0,Y 358.197,Z 654.157,A -85,B 0,C 180,E1 -14887.373,E2 -14887.373} C_VEL
LIN {X 0,Y 361.502,Z 566.266,A -85,B 0,C 180,E1 -14889.143,E2 -14889.143} C_VEL
LIN {X 0,Y 362.425,Z 539.192,A -85,B 0,C 180,E1 -14889.703,E2 -14889.703} C_VEL
LIN {X 0,Y 361.252,Z 534.812,A -85,B 0,C 180,E1 -14889.967,E2 -14889.967} C_VEL
LIN {X 0,Y 352.884,Z 517.181,A -85,B 0,C 180,E1 -14891.574,E2 -14891.574} C_VEL
LIN {X 0,Y 344.144,Z 500.663,A -85,B 0,C 180,E1 -14893.329,E2 -14893.329} C_VEL
LIN {X 0,Y 335.428,Z 485.728,A -85,B 0,C 180,E1 -14895.18,E2 -14895.18} C_VEL
LIN {X 0,Y 331.596,Z 479.707,A -85,B 0,C 180,E1 -14896.029,E2 -14896.029} C_VEL
LIN {X 0,Y 329.467,Z 475.897,A -85,B 0,C 180,E1 -14896.585,E2 -14896.585} C_VEL
LIN {X 0,Y 326.684,Z 467.348,A -85,B 0,C 180,E1 -14899.699,E2 -14899.699} C_VEL
LIN {X 0,Y 326.615,Z 467.022,A -85,B 0,C 180,E1 -14900.332,E2 -14900.332} C_VEL
LIN {X 0,Y 326.628,Z 467.039,A -85,B 0,C 180,E1 -14902.953,E2 -14902.953} C_VEL
LIN {X 0,Y 326.604,Z 467.019,A -85,B 0,C 180,E1 -14905.98,E2 -14905.98} C_VEL
LIN {X 0,Y 326.636,Z 467.02,A -85,B 0,C 180,E1 -14909.387,E2 -14909.387} C_VEL
LIN {X 0,Y 326.679,Z 466.995,A -85,B 0,C 180,E1 -14913.142,E2 -14913.142} C_VEL
LIN {X 0,Y 326.643,Z 467.048,A -85,B 0,C 180,E1 -14915.87,E2 -14915.87} C_VEL
LIN {X 0,Y 326.651,Z 466.974,A -85,B 0,C 180,E1 -14919.864,E2 -14919.864} C_VEL
LIN {X 0,Y 326.692,Z 467.009,A -85,B 0,C 180,E1 -14922.472,E2 -14922.472} C_VEL
LIN {X 0,Y 326.752,Z 467.014,A -85,B 0,C 180,E1 -14926.314,E2 -14926.314} C_VEL
LIN {X 0,Y 326.799,Z 467.017,A -85,B 0,C 180,E1 -14930.093,E2 -14930.093} C_VEL
LIN {X 0,Y 326.985,Z 467.004,A -85,B 0,C 180,E1 -14933.83,E2 -14933.83} C_VEL
LIN {X 0,Y 327.04,Z 466.986,A -85,B 0,C 180,E1 -14937.536,E2 -14937.536} C_VEL
LIN {X 0,Y 327.173,Z 466.97,A -85,B 0,C 180,E1 -14940,E2 -14940} C_VEL
LIN {X 0,Y 327.041,Z 466.98,A -85,B 0,C 180,E1 -14942.463,E2 -14942.463} C_VEL
LIN {X 0,Y 326.958,Z 466.985,A -85,B 0,C 180,E1 -14946.608,E2 -14946.608} C_VEL
LIN {X 0,Y 326.908,Z 467.011,A -85,B 0,C 180,E1 -14948.655,E2 -14948.655} C_VEL
LIN {X 0,Y 326.726,Z 467.025,A -85,B 0,C 180,E1 -14952.421,E2 -14952.421} C_VEL
LIN {X 0,Y 326.747,Z 467.019,A -85,B 0,C 180,E1 -14954.957,E2 -14954.957} C_VEL
LIN {X 0,Y 326.726,Z 467.033,A -85,B 0,C 180,E1 -14958.838,E2 -14958.838} C_VEL
LIN {X 0,Y 326.598,Z 467.054,A -85,B 0,C 180,E1 -14962.789,E2 -14962.789} C_VEL
LIN {X 0,Y 326.683,Z 466.988,A -85,B 0,C 180,E1 -14965.484,E2 -14965.484} C_VEL
LIN {X 0,Y 326.654,Z 467.036,A -85,B 0,C 180,E1 -14969.659,E2 -14969.659} C_VEL
LIN {X 0,Y 326.6,Z 466.998,A -85,B 0,C 180,E1 -14974.02,E2 -14974.02} C_VEL
LIN {X 0,Y 326.626,Z 467.051,A -85,B 0,C 180,E1 -14977.24,E2 -14977.24} C_VEL
LIN {X 0,Y 326.63,Z 467.051,A -85,B 0,C 180,E1 -14980.203,E2 -14980.203} C_VEL
LIN {X 0,Y 326.631,Z 467.05,A -85,B 0,C 180,E1 -14984.135,E2 -14984.135} C_VEL
LIN {X 0,Y 326.669,Z 467.527,A -85,B 0,C 180,E1 -14984.937,E2 -14984.937} C_VEL
LIN {X 0,Y 327.298,Z 469.326,A -85,B 0,C 180,E1 -14985.474,E2 -14985.474} C_VEL
LIN {X 0,Y 329.125,Z 471.622,A -85,B 0,C 180,E1 -14986.239,E2 -14986.239} C_VEL
LIN {X 0,Y 331.477,Z 473.16,A -85,B 0,C 180,E1 -14987.177,E2 -14987.177} C_VEL
LIN {X 0,Y 333.27,Z 476.185,A -85,B 0,C 180,E1 -14987.974,E2 -14987.974} C_VEL
LIN {X 0,Y 335.963,Z 478.487,A -85,B 0,C 180,E1 -14989.108,E2 -14989.108} C_VEL
LIN {X 0,Y 336.903,Z 479.251,A -85,B 0,C 180,E1 -14989.49,E2 -14989.49} C_VEL
LIN {X 0,Y 338.868,Z 482.194,A -85,B 0,C 180,E1 -14990.408,E2 -14990.408} C_VEL
LIN {X 0,Y 341.597,Z 484.394,A -85,B 0,C 180,E1 -14991.583,E2 -14991.583} C_VEL
LIN {X 0,Y 342.411,Z 485.204,A -85,B 0,C 180,E1 -14991.947,E2 -14991.947} C_VEL
LIN {X 0,Y 344.532,Z 488.152,A -85,B 0,C 180,E1 -14992.948,E2 -14992.948} C_VEL
LIN {X 0,Y 348.003,Z 490.967,A -85,B 0,C 180,E1 -14994.525,E2 -14994.525} C_VEL
LIN {X 0,Y 350.416,Z 494.206,A -85,B 0,C 180,E1 -14995.717,E2 -14995.717} C_VEL
LIN {X 0,Y 353.576,Z 496.655,A -85,B 0,C 180,E1 -14997.231,E2 -14997.231} C_VEL
LIN {X 0,Y 356.806,Z 500.651,A -85,B 0,C 180,E1 -14998.93,E2 -14998.93} C_VEL
LIN {X 0,Y 359.894,Z 502.828,A -85,B 0,C 180,E1 -15000.519,E2 -15000.519} C_VEL
LIN {X 0,Y 363.043,Z 506.712,A -85,B 0,C 180,E1 -15002.316,E2 -15002.316} C_VEL
LIN {X 0,Y 366.355,Z 509.142,A -85,B 0,C 180,E1 -15004.211,E2 -15004.211} C_VEL
LIN {X 0,Y 369.401,Z 513.031,A -85,B 0,C 180,E1 -15006.203,E2 -15006.203} C_VEL
LIN {X 0,Y 372.478,Z 515.255,A -85,B 0,C 180,E1 -15008.202,E2 -15008.202} C_VEL
LIN {X 0,Y 373.58,Z 515.968,A -85,B 0,C 180,E1 -15008.987,E2 -15008.987} C_VEL
LIN {X 0,Y 375.794,Z 518.958,A -85,B 0,C 180,E1 -15010.718,E2 -15010.718} C_VEL
LIN {X 0,Y 378.655,Z 521.27,A -85,B 0,C 180,E1 -15013.074,E2 -15013.074} C_VEL
LIN {X 0,Y 380.916,Z 522.61,A -85,B 0,C 180,E1 -15015.099,E2 -15015.099} C_VEL
LIN {X 0,Y 382.574,Z 525.128,A -85,B 0,C 180,E1 -15017.008,E2 -15017.008} C_VEL
LIN {X 0,Y 384.44,Z 526.914,A -85,B 0,C 180,E1 -15019.307,E2 -15019.307} C_VEL
LIN {X 0,Y 386.26,Z 527.938,A -85,B 0,C 180,E1 -15022.082,E2 -15022.082} C_VEL
LIN {X 0,Y 387.538,Z 528.612,A -85,B 0,C 180,E1 -15024.798,E2 -15024.798} C_VEL
LIN {X 0,Y 388.152,Z 528.945,A -85,B 0,C 180,E1 -15026.886,E2 -15026.886} C_VEL
LIN {X 0,Y 388.446,Z 529.196,A -85,B 0,C 180,E1 -15028.963,E2 -15028.963} C_VEL
LIN {X 0,Y 388.446,Z 529.199,A -85,B 0,C 180,E1 -15031.037,E2 -15031.037} C_VEL
LIN {X 0,Y 388.152,Z 528.946,A -85,B 0,C 180,E1 -15033.114,E2 -15033.114} C_VEL
LIN {X 0,Y 387.408,Z 528.491,A -85,B 0,C 180,E1 -15035.553,E2 -15035.553} C_VEL
LIN {X 0,Y 386,Z 527.791,A -85,B 0,C 180,E1 -15038.375,E2 -15038.375} C_VEL
LIN {X 0,Y 384.319,Z 526.804,A -85,B 0,C 180,E1 -15040.856,E2 -15040.856} C_VEL
LIN {X 0,Y 382.547,Z 525.087,A -85,B 0,C 180,E1 -15043.025,E2 -15043.025} C_VEL
LIN {X 0,Y 380.434,Z 522.16,A -85,B 0,C 180,E1 -15045.361,E2 -15045.361} C_VEL
LIN {X 0,Y 377.526,Z 520.499,A -85,B 0,C 180,E1 -15047.884,E2 -15047.884} C_VEL
LIN {X 0,Y 375.252,Z 518.313,A -85,B 0,C 180,E1 -15049.701,E2 -15049.701} C_VEL
LIN {X 0,Y 373.287,Z 515.616,A -85,B 0,C 180,E1 -15051.232,E2 -15051.232} C_VEL
LIN {X 0,Y 370.332,Z 513.853,A -85,B 0,C 180,E1 -15053.215,E2 -15053.215} C_VEL
LIN {X 0,Y 367.484,Z 510.706,A -85,B 0,C 180,E1 -15055.056,E2 -15055.056} C_VEL
LIN {X 0,Y 366.361,Z 509.124,A -85,B 0,C 180,E1 -15055.789,E2 -15055.789} C_VEL
LIN {X 0,Y 363.042,Z 506.745,A -85,B 0,C 180,E1 -15057.684,E2 -15057.684} C_VEL
LIN {X 0,Y 360.273,Z 503.206,A -85,B 0,C 180,E1 -15059.277,E2 -15059.277} C_VEL
LIN {X 0,Y 356.678,Z 500.513,A -85,B 0,C 180,E1 -15061.137,E2 -15061.137} C_VEL
LIN {X 0,Y 354.092,Z 497.264,A -85,B 0,C 180,E1 -15062.498,E2 -15062.498} C_VEL
LIN {X 0,Y 353.144,Z 496.427,A -85,B 0,C 180,E1 -15062.979,E2 -15062.979} C_VEL
LIN {X 0,Y 349.877,Z 493.585,A -85,B 0,C 180,E1 -15064.557,E2 -15064.557} C_VEL
LIN {X 0,Y 347.731,Z 490.614,A -85,B 0,C 180,E1 -15065.61,E2 -15065.61} C_VEL
LIN {X 0,Y 344.531,Z 488.169,A -85,B 0,C 180,E1 -15067.052,E2 -15067.052} C_VEL
LIN {X 0,Y 342.229,Z 484.884,A -85,B 0,C 180,E1 -15068.141,E2 -15068.141} C_VEL
LIN {X 0,Y 338.958,Z 482.304,A -85,B 0,C 180,E1 -15069.553,E2 -15069.553} C_VEL
LIN {X 0,Y 336.995,Z 479.451,A -85,B 0,C 180,E1 -15070.465,E2 -15070.465} C_VEL
LIN {X 0,Y 336.389,Z 478.709,A -85,B 0,C 180,E1 -15070.724,E2 -15070.724} C_VEL
LIN {X 0,Y 333.599,Z 476.564,A -85,B 0,C 180,E1 -15071.885,E2 -15071.885} C_VEL
LIN {X 0,Y 331.746,Z 473.737,A -85,B 0,C 180,E1 -15072.695,E2 -15072.695} C_VEL
LIN {X 0,Y 331.204,Z 472.847,A -85,B 0,C 180,E1 -15072.939,E2 -15072.939} C_VEL
LIN {X 0,Y 328.718,Z 471.265,A -85,B 0,C 180,E1 -15073.921,E2 -15073.921} C_VEL
LIN {X 0,Y 327.2,Z 469.129,A -85,B 0,C 180,E1 -15074.58,E2 -15074.58} C_VEL
LIN {X 0,Y 326.669,Z 467.527,A -85,B 0,C 180,E1 -15075.063,E2 -15075.063} C_VEL
LIN {X 0,Y 326.631,Z 467.05,A -85,B 0,C 180,E1 -15075.865,E2 -15075.865} C_VEL
LIN {X 0,Y 326.63,Z 467.051,A -85,B 0,C 180,E1 -15079.797,E2 -15079.797} C_VEL
LIN {X 0,Y 326.629,Z 467.048,A -85,B 0,C 180,E1 -15082.954,E2 -15082.954} C_VEL
LIN {X 0,Y 326.6,Z 466.998,A -85,B 0,C 180,E1 -15085.98,E2 -15085.98} C_VEL
LIN {X 0,Y 326.654,Z 467.036,A -85,B 0,C 180,E1 -15090.341,E2 -15090.341} C_VEL
LIN {X 0,Y 326.683,Z 466.987,A -85,B 0,C 180,E1 -15094.516,E2 -15094.516} C_VEL
LIN {X 0,Y 326.613,Z 467.041,A -85,B 0,C 180,E1 -15098.543,E2 -15098.543} C_VEL
LIN {X 0,Y 326.738,Z 467.031,A -85,B 0,C 180,E1 -15101.178,E2 -15101.178} C_VEL
LIN {X 0,Y 326.75,Z 467.021,A -85,B 0,C 180,E1 -15105.283,E2 -15105.283} C_VEL
LIN {X 0,Y 326.101,Z 467.114,A -85,B 0,C 180,E1 -15106.312,E2 -15106.312} C_VEL
LIN {X 0,Y 323.235,Z 467.462,A -85,B 0,C 180,E1 -15107.986,E2 -15107.986} C_VEL
LIN {X 0,Y 320.828,Z 467.756,A -85,B 0,C 180,E1 -15109.343,E2 -15109.343} C_VEL
LIN {X 0,Y 319.844,Z 467.887,A -85,B 0,C 180,E1 -15110.394,E2 -15110.394} C_VEL
LIN {X 0,Y 319.791,Z 467.892,A -85,B 0,C 180,E1 -15110.749,E2 -15110.749} C_VEL
LIN {X 0,Y 319.939,Z 467.861,A -85,B 0,C 180,E1 -15113.695,E2 -15113.695} C_VEL
LIN {X 0,Y 319.985,Z 467.861,A -85,B 0,C 180,E1 -15117.483,E2 -15117.483} C_VEL
LIN {X 0,Y 320.125,Z 467.849,A -85,B 0,C 180,E1 -15120,E2 -15120} C_VEL
LIN {X 0,Y 319.984,Z 467.864,A -85,B 0,C 180,E1 -15122.518,E2 -15122.518} C_VEL
LIN {X 0,Y 319.939,Z 467.88,A -85,B 0,C 180,E1 -15126.306,E2 -15126.306} C_VEL
LIN {X 0,Y 319.831,Z 467.873,A -85,B 0,C 180,E1 -15128.849,E2 -15128.849} C_VEL
LIN {X 0,Y 319.674,Z 467.896,A -85,B 0,C 180,E1 -15132.7,E2 -15132.7} C_VEL
LIN {X 0,Y 319.693,Z 467.91,A -85,B 0,C 180,E1 -15135.296,E2 -15135.296} C_VEL
LIN {X 0,Y 319.645,Z 467.849,A -85,B 0,C 180,E1 -15139.257,E2 -15139.257} C_VEL
LIN {X 0,Y 319.554,Z 467.916,A -85,B 0,C 180,E1 -15143.321,E2 -15143.321} C_VEL
LIN {X 0,Y 319.613,Z 467.891,A -85,B 0,C 180,E1 -15146.09,E2 -15146.09} C_VEL
LIN {X 0,Y 319.584,Z 467.866,A -85,B 0,C 180,E1 -15148.934,E2 -15148.934} C_VEL
LIN {X 0,Y 319.534,Z 467.933,A -85,B 0,C 180,E1 -15151.862,E2 -15151.862} C_VEL
LIN {X 0,Y 319.575,Z 467.891,A -85,B 0,C 180,E1 -15155.544,E2 -15155.544} C_VEL
LIN {X 0,Y 319.631,Z 468.05,A -85,B 0,C 180,E1 -15159.107,E2 -15159.107} C_VEL
LIN {X 0,Y 322.05,Z 475.538,A -85,B 0,C 180,E1 -15162.004,E2 -15162.004} C_VEL
LIN {X 0,Y 325.336,Z 480.811,A -85,B 0,C 180,E1 -15162.86,E2 -15162.86} C_VEL
LIN {X 0,Y 330.294,Z 489.021,A -85,B 0,C 180,E1 -15164.023,E2 -15164.023} C_VEL
LIN {X 0,Y 335.317,Z 497.258,A -85,B 0,C 180,E1 -15165.142,E2 -15165.142} C_VEL
LIN {X 0,Y 343.101,Z 511.293,A -85,B 0,C 180,E1 -15166.807,E2 -15166.807} C_VEL
LIN {X 0,Y 351.971,Z 528.935,A -85,B 0,C 180,E1 -15168.608,E2 -15168.608} C_VEL
LIN {X 0,Y 356.605,Z 539.132,A -85,B 0,C 180,E1 -15169.521,E2 -15169.521} C_VEL
LIN {X 0,Y 356.998,Z 541.165,A -85,B 0,C 180,E1 -15169.627,E2 -15169.627} C_VEL
LIN {X 0,Y 351.636,Z 679.024,A -85,B 0,C 180,E1 -15172.441,E2 -15172.441} C_VEL
LIN {X 0,Y 350.453,Z 698.69,A -85,B 0,C 180,E1 -15172.925,E2 -15172.925} C_VEL
LIN {X 0,Y 348.965,Z 713.468,A -85,B 0,C 180,E1 -15173.462,E2 -15173.462} C_VEL
LIN {X 0,Y 347.369,Z 726.329,A -85,B 0,C 180,E1 -15174.076,E2 -15174.076} C_VEL
LIN {X 0,Y 345.599,Z 738.578,A -85,B 0,C 180,E1 -15174.8,E2 -15174.8} C_VEL
LIN {X 0,Y 343.341,Z 751.771,A -85,B 0,C 180,E1 -15175.744,E2 -15175.744} C_VEL
LIN {X 0,Y 341.181,Z 763.414,A -85,B 0,C 180,E1 -15176.74,E2 -15176.74} C_VEL
LIN {X 0,Y 338.766,Z 774.937,A -85,B 0,C 180,E1 -15177.886,E2 -15177.886} C_VEL
LIN {X 0,Y 336.014,Z 787.251,A -85,B 0,C 180,E1 -15179.33,E2 -15179.33} C_VEL
LIN {X 0,Y 333.347,Z 798.217,A -85,B 0,C 180,E1 -15180.821,E2 -15180.821} C_VEL
LIN {X 0,Y 331.229,Z 806.902,A -85,B 0,C 180,E1 -15182.174,E2 -15182.174} C_VEL
LIN {X 0,Y 328.898,Z 816.221,A -85,B 0,C 180,E1 -15183.827,E2 -15183.827} C_VEL
LIN {X 0,Y 326.414,Z 826.072,A -85,B 0,C 180,E1 -15185.853,E2 -15185.853} C_VEL
LIN {X 0,Y 324.426,Z 833.965,A -85,B 0,C 180,E1 -15187.723,E2 -15187.723} C_VEL
LIN {X 0,Y 322.818,Z 840.932,A -85,B 0,C 180,E1 -15189.615,E2 -15189.615} C_VEL
LIN {X 0,Y 321.473,Z 847.076,A -85,B 0,C 180,E1 -15191.519,E2 -15191.519} C_VEL
LIN {X 0,Y 319.989,Z 854.023,A -85,B 0,C 180,E1 -15194.066,E2 -15194.066} C_VEL
LIN {X 0,Y 319.243,Z 858.497,A -85,B 0,C 180,E1 -15195.986,E2 -15195.986} C_VEL
LIN {X 0,Y 318.407,Z 863.395,A -85,B 0,C 180,E1 -15198.542,E2 -15198.542} C_VEL
LIN {X 0,Y 317.961,Z 867.247,A -85,B 0,C 180,E1 -15201.099,E2 -15201.099} C_VEL
LIN {X 0,Y 317.85,Z 870.1,A -85,B 0,C 180,E1 -15203.653,E2 -15203.653} C_VEL
LIN {X 0,Y 317.776,Z 871.983,A -85,B 0,C 180,E1 -15206.196,E2 -15206.196} C_VEL
LIN {X 0,Y 317.744,Z 872.657,A -85,B 0,C 180,E1 -15207.465,E2 -15207.465} C_VEL
LIN {X 0,Y 317.728,Z 873.129,A -85,B 0,C 180,E1 -15210,E2 -15210} C_VEL
LIN {X 0,Y 317.744,Z 872.657,A -85,B 0,C 180,E1 -15212.535,E2 -15212.535} C_VEL
LIN {X 0,Y 317.808,Z 870.714,A -85,B 0,C 180,E1 -15215.659,E2 -15215.659} C_VEL
LIN {X 0,Y 317.864,Z 868.849,A -85,B 0,C 180,E1 -15217.623,E2 -15217.623} C_VEL
LIN {X 0,Y 318.242,Z 864.434,A -85,B 0,C 180,E1 -15220.819,E2 -15220.819} C_VEL
LIN {X 0,Y 318.726,Z 861.068,A -85,B 0,C 180,E1 -15222.738,E2 -15222.738} C_VEL
LIN {X 0,Y 319.454,Z 856.884,A -85,B 0,C 180,E1 -15224.751,E2 -15224.751} C_VEL
LIN {X 0,Y 320.668,Z 850.709,A -85,B 0,C 180,E1 -15227.21,E2 -15227.21} C_VEL
LIN {X 0,Y 322.321,Z 843.039,A -85,B 0,C 180,E1 -15229.753,E2 -15229.753} C_VEL
LIN {X 0,Y 323.817,Z 836.383,A -85,B 0,C 180,E1 -15231.651,E2 -15231.651} C_VEL
LIN {X 0,Y 325.719,Z 828.831,A -85,B 0,C 180,E1 -15233.526,E2 -15233.526} C_VEL
LIN {X 0,Y 327.963,Z 820.248,A -85,B 0,C 180,E1 -15235.377,E2 -15235.377} C_VEL
LIN {X 0,Y 330.324,Z 810.453,A -85,B 0,C 180,E1 -15237.221,E2 -15237.221} C_VEL
LIN {X 0,Y 332.861,Z 800.23,A -85,B 0,C 180,E1 -15238.88,E2 -15238.88} C_VEL
LIN {X 0,Y 335.152,Z 790.808,A -85,B 0,C 180,E1 -15240.216,E2 -15240.216} C_VEL
LIN {X 0,Y 337.619,Z 780.158,A -85,B 0,C 180,E1 -15241.534,E2 -15241.534} C_VEL
LIN {X 0,Y 340.225,Z 767.912,A -85,B 0,C 180,E1 -15242.836,E2 -15242.836} C_VEL
LIN {X 0,Y 342.39,Z 756.997,A -85,B 0,C 180,E1 -15243.832,E2 -15243.832} C_VEL
LIN {X 0,Y 344.69,Z 744.266,A -85,B 0,C 180,E1 -15244.812,E2 -15244.812} C_VEL
LIN {X 0,Y 346.515,Z 732.255,A -85,B 0,C 180,E1 -15245.597,E2 -15245.597} C_VEL
LIN {X 0,Y 348.413,Z 718.287,A -85,B 0,C 180,E1 -15246.323,E2 -15246.323} C_VEL
LIN {X 0,Y 349.944,Z 704.537,A -85,B 0,C 180,E1 -15246.875,E2 -15246.875} C_VEL
LIN {X 0,Y 351.01,Z 691.233,A -85,B 0,C 180,E1 -15247.276,E2 -15247.276} C_VEL
LIN {X 0,Y 352.565,Z 653.947,A -85,B 0,C 180,E1 -15248.075,E2 -15248.075} C_VEL
LIN {X 0,Y 355.816,Z 571.841,A -85,B 0,C 180,E1 -15249.743,E2 -15249.743} C_VEL
LIN {X 0,Y 356.913,Z 540.78,A -85,B 0,C 180,E1 -15250.395,E2 -15250.395} C_VEL
LIN {X 0,Y 355.891,Z 537.493,A -85,B 0,C 180,E1 -15250.619,E2 -15250.619} C_VEL
LIN {X 0,Y 348.158,Z 521.16,A -85,B 0,C 180,E1 -15252.154,E2 -15252.154} C_VEL
LIN {X 0,Y 339.934,Z 505.422,A -85,B 0,C 180,E1 -15253.861,E2 -15253.861} C_VEL
LIN {X 0,Y 331.278,Z 490.472,A -85,B 0,C 180,E1 -15255.758,E2 -15255.758} C_VEL
LIN {X 0,Y 324.804,Z 480.137,A -85,B 0,C 180,E1 -15257.262,E2 -15257.262} C_VEL
LIN {X 0,Y 321.989,Z 475.477,A -85,B 0,C 180,E1 -15258.02,E2 -15258.02} C_VEL
LIN {X 0,Y 319.631,Z 468.056,A -85,B 0,C 180,E1 -15260.893,E2 -15260.893} C_VEL
LIN {X 0,Y 319.555,Z 467.891,A -85,B 0,C 180,E1 -15265.123,E2 -15265.123} C_VEL
LIN {X 0,Y 319.57,Z 467.907,A -85,B 0,C 180,E1 -15269.056,E2 -15269.056} C_VEL
LIN {X 0,Y 319.603,Z 467.866,A -85,B 0,C 180,E1 -15272.498,E2 -15272.498} C_VEL
LIN {X 0,Y 319.598,Z 467.924,A -85,B 0,C 180,E1 -15275.303,E2 -15275.303} C_VEL
LIN {X 0,Y 319.595,Z 467.852,A -85,B 0,C 180,E1 -15279.4,E2 -15279.4} C_VEL
LIN {X 0,Y 319.652,Z 467.872,A -85,B 0,C 180,E1 -15282.073,E2 -15282.073} C_VEL
LIN {X 0,Y 319.725,Z 467.891,A -85,B 0,C 180,E1 -15286.007,E2 -15286.007} C_VEL
LIN {X 0,Y 319.746,Z 467.898,A -85,B 0,C 180,E1 -15289.872,E2 -15289.872} C_VEL
LIN {X 0,Y 319.907,Z 467.87,A -85,B 0,C 180,E1 -15292.425,E2 -15292.425} C_VEL
LIN {X 0,Y 319.741,Z 467.9,A -85,B 0,C 180,E1 -15294.956,E2 -15294.956} C_VEL
LIN {X 0,Y 319.984,Z 467.863,A -85,B 0,C 180,E1 -15297.482,E2 -15297.482} C_VEL
LIN {X 0,Y 320.125,Z 467.847,A -85,B 0,C 180,E1 -15300,E2 -15300} C_VEL
LIN {X 0,Y 319.985,Z 467.859,A -85,B 0,C 180,E1 -15302.517,E2 -15302.517} C_VEL
LIN {X 0,Y 319.92,Z 467.861,A -85,B 0,C 180,E1 -15306.597,E2 -15306.597} C_VEL
LIN {X 0,Y 319.835,Z 467.891,A -85,B 0,C 180,E1 -15308.848,E2 -15308.848} C_VEL
LIN {X 0,Y 319.674,Z 467.906,A -85,B 0,C 180,E1 -15312.7,E2 -15312.7} C_VEL
LIN {X 0,Y 319.692,Z 467.894,A -85,B 0,C 180,E1 -15315.295,E2 -15315.295} C_VEL
LIN {X 0,Y 319.645,Z 467.91,A -85,B 0,C 180,E1 -15319.256,E2 -15319.256} C_VEL
LIN {X 0,Y 319.554,Z 467.926,A -85,B 0,C 180,E1 -15323.32,E2 -15323.32} C_VEL
LIN {X 0,Y 319.612,Z 467.86,A -85,B 0,C 180,E1 -15326.09,E2 -15326.09} C_VEL
LIN {X 0,Y 319.582,Z 467.893,A -85,B 0,C 180,E1 -15328.934,E2 -15328.934} C_VEL
LIN {X 0,Y 319.526,Z 467.907,A -85,B 0,C 180,E1 -15331.862,E2 -15331.862} C_VEL
LIN {X 0,Y 319.574,Z 467.886,A -85,B 0,C 180,E1 -15335.543,E2 -15335.543} C_VEL
LIN {X 0,Y 319.596,Z 467.926,A -85,B 0,C 180,E1 -15338.004,E2 -15338.004} C_VEL
LIN {X 0,Y 319.591,Z 467.927,A -85,B 0,C 180,E1 -15341.612,E2 -15341.612} C_VEL
LIN {X 0,Y 319.575,Z 468.058,A -85,B 0,C 180,E1 -15342.422,E2 -15342.422} C_VEL
LIN {X 0,Y 319.886,Z 469.304,A -85,B 0,C 180,E1 -15342.927,E2 -15342.927} C_VEL
LIN {X 0,Y 321.169,Z 471.608,A -85,B 0,C 180,E1 -15343.468,E2 -15343.468} C_VEL
LIN {X 0,Y 323.697,Z 473.556,A -85,B 0,C 180,E1 -15344.405,E2 -15344.405} C_VEL
LIN {X 0,Y 324.622,Z 474.658,A -85,B 0,C 180,E1 -15344.778,E2 -15344.778} C_VEL
LIN {X 0,Y 326.554,Z 477.491,A -85,B 0,C 180,E1 -15345.607,E2 -15345.607} C_VEL
LIN {X 0,Y 329.221,Z 479.468,A -85,B 0,C 180,E1 -15346.652,E2 -15346.652} C_VEL
LIN {X 0,Y 331.895,Z 483.264,A -85,B 0,C 180,E1 -15347.828,E2 -15347.828} C_VEL
LIN {X 0,Y 334.982,Z 485.844,A -85,B 0,C 180,E1 -15349.113,E2 -15349.113} C_VEL
LIN {X 0,Y 337.331,Z 489.03,A -85,B 0,C 180,E1 -15350.168,E2 -15350.168} C_VEL
LIN {X 0,Y 340.603,Z 491.755,A -85,B 0,C 180,E1 -15351.576,E2 -15351.576} C_VEL
LIN {X 0,Y 343.123,Z 495.045,A -85,B 0,C 180,E1 -15352.741,E2 -15352.741} C_VEL
LIN {X 0,Y 346.434,Z 497.781,A -85,B 0,C 180,E1 -15354.238,E2 -15354.238} C_VEL
LIN {X 0,Y 349.225,Z 501.272,A -85,B 0,C 180,E1 -15355.598,E2 -15355.598} C_VEL
LIN {X 0,Y 352.614,Z 504.075,A -85,B 0,C 180,E1 -15357.234,E2 -15357.234} C_VEL
LIN {X 0,Y 355.542,Z 507.554,A -85,B 0,C 180,E1 -15358.757,E2 -15358.757} C_VEL
LIN {X 0,Y 358.999,Z 510.232,A -85,B 0,C 180,E1 -15360.549,E2 -15360.549} C_VEL
LIN {X 0,Y 361.812,Z 513.639,A -85,B 0,C 180,E1 -15362.15,E2 -15362.15} C_VEL
LIN {X 0,Y 365.467,Z 516.423,A -85,B 0,C 180,E1 -15364.235,E2 -15364.235} C_VEL
LIN {X 0,Y 368.178,Z 519.902,A -85,B 0,C 180,E1 -15366.001,E2 -15366.001} C_VEL
LIN {X 0,Y 371.04,Z 522.053,A -85,B 0,C 180,E1 -15367.861,E2 -15367.861} C_VEL
LIN {X 0,Y 372.479,Z 523.015,A -85,B 0,C 180,E1 -15368.85,E2 -15368.85} C_VEL
LIN {X 0,Y 374.619,Z 525.825,A -85,B 0,C 180,E1 -15370.51,E2 -15370.51} C_VEL
LIN {X 0,Y 377.534,Z 528.185,A -85,B 0,C 180,E1 -15372.869,E2 -15372.869} C_VEL
LIN {X 0,Y 379.925,Z 529.642,A -85,B 0,C 180,E1 -15374.991,E2 -15374.991} C_VEL
LIN {X 0,Y 381.502,Z 532.005,A -85,B 0,C 180,E1 -15376.777,E2 -15376.777} C_VEL
LIN {X 0,Y 383.417,Z 533.866,A -85,B 0,C 180,E1 -15379.117,E2 -15379.117} C_VEL
LIN {X 0,Y 385.12,Z 534.813,A -85,B 0,C 180,E1 -15381.606,E2 -15381.606} C_VEL
LIN {X 0,Y 386.533,Z 535.536,A -85,B 0,C 180,E1 -15384.433,E2 -15384.433} C_VEL
LIN {X 0,Y 387.285,Z 535.991,A -85,B 0,C 180,E1 -15386.879,E2 -15386.879} C_VEL
LIN {X 0,Y 387.581,Z 536.232,A -85,B 0,C 180,E1 -15388.961,E2 -15388.961} C_VEL
LIN {X 0,Y 387.581,Z 536.235,A -85,B 0,C 180,E1 -15391.039,E2 -15391.039} C_VEL
LIN {X 0,Y 387.214,Z 535.97,A -85,B 0,C 180,E1 -15393.392,E2 -15393.392} C_VEL
LIN {X 0,Y 386.533,Z 535.538,A -85,B 0,C 180,E1 -15395.566,E2 -15395.566} C_VEL
LIN {X 0,Y 385.117,Z 534.835,A -85,B 0,C 180,E1 -15398.395,E2 -15398.395} C_VEL
LIN {X 0,Y 383.422,Z 533.848,A -85,B 0,C 180,E1 -15400.882,E2 -15400.882} C_VEL
LIN {X 0,Y 381.668,Z 532.201,A -85,B 0,C 180,E1 -15403.021,E2 -15403.021} C_VEL
LIN {X 0,Y 379.817,Z 529.455,A -85,B 0,C 180,E1 -15405.12,E2 -15405.12} C_VEL
LIN {X 0,Y 376.633,Z 527.564,A -85,B 0,C 180,E1 -15407.889,E2 -15407.889} C_VEL
LIN {X 0,Y 374.101,Z 525.221,A -85,B 0,C 180,E1 -15409.897,E2 -15409.897} C_VEL
LIN {X 0,Y 372.107,Z 522.539,A -85,B 0,C 180,E1 -15411.433,E2 -15411.433} C_VEL
LIN {X 0,Y 368.824,Z 520.497,A -85,B 0,C 180,E1 -15413.587,E2 -15413.587} C_VEL
LIN {X 0,Y 365.973,Z 517.24,A -85,B 0,C 180,E1 -15415.427,E2 -15415.427} C_VEL
LIN {X 0,Y 365.044,Z 515.983,A -85,B 0,C 180,E1 -15416.034,E2 -15416.034} C_VEL
LIN {X 0,Y 361.629,Z 513.497,A -85,B 0,C 180,E1 -15417.951,E2 -15417.951} C_VEL
LIN {X 0,Y 358.79,Z 509.943,A -85,B 0,C 180,E1 -15419.569,E2 -15419.569} C_VEL
LIN {X 0,Y 355.195,Z 507.218,A -85,B 0,C 180,E1 -15421.427,E2 -15421.427} C_VEL
LIN {X 0,Y 352.414,Z 503.758,A -85,B 0,C 180,E1 -15422.876,E2 -15422.876} C_VEL
LIN {X 0,Y 348.529,Z 500.566,A -85,B 0,C 180,E1 -15424.732,E2 -15424.732} C_VEL
LIN {X 0,Y 345.909,Z 497.213,A -85,B 0,C 180,E1 -15426.013,E2 -15426.013} C_VEL
LIN {X 0,Y 342.465,Z 494.328,A -85,B 0,C 180,E1 -15427.562,E2 -15427.562} C_VEL
LIN {X 0,Y 340.166,Z 491.216,A -85,B 0,C 180,E1 -15428.628,E2 -15428.628} C_VEL
LIN {X 0,Y 337.126,Z 488.805,A -85,B 0,C 180,E1 -15429.923,E2 -15429.923} C_VEL
LIN {X 0,Y 334.885,Z 485.674,A -85,B 0,C 180,E1 -15430.931,E2 -15430.931} C_VEL
LIN {X 0,Y 331.48,Z 482.797,A -85,B 0,C 180,E1 -15432.344,E2 -15432.344} C_VEL
LIN {X 0,Y 329.312,Z 479.521,A -85,B 0,C 180,E1 -15433.311,E2 -15433.311} C_VEL
LIN {X 0,Y 326.671,Z 477.649,A -85,B 0,C 180,E1 -15434.343,E2 -15434.343} C_VEL
LIN {X 0,Y 324.686,Z 474.775,A -85,B 0,C 180,E1 -15435.194,E2 -15435.194} C_VEL
LIN {X 0,Y 323.895,Z 473.672,A -85,B 0,C 180,E1 -15435.52,E2 -15435.52} C_VEL
LIN {X 0,Y 321.265,Z 471.713,A -85,B 0,C 180,E1 -15436.495,E2 -15436.495} C_VEL
LIN {X 0,Y 319.801,Z 469.018,A -85,B 0,C 180,E1 -15437.152,E2 -15437.152} C_VEL
LIN {X 0,Y 319.577,Z 467.994,A -85,B 0,C 180,E1 -15437.671,E2 -15437.671} C_VEL
LIN {X 0,Y 319.581,Z 467.928,A -85,B 0,C 180,E1 -15440.377,E2 -15440.377} C_VEL
LIN {X 0,Y 319.555,Z 467.909,A -85,B 0,C 180,E1 -15443.573,E2 -15443.573} C_VEL
LIN {X 0,Y 319.57,Z 467.876,A -85,B 0,C 180,E1 -15446.686,E2 -15446.686} C_VEL
LIN {X 0,Y 319.585,Z 467.928,A -85,B 0,C 180,E1 -15449.616,E2 -15449.616} C_VEL
LIN {X 0,Y 319.601,Z 467.864,A -85,B 0,C 180,E1 -15452.498,E2 -15452.498} C_VEL
LIN {X 0,Y 319.596,Z 467.883,A -85,B 0,C 180,E1 -15455.304,E2 -15455.304} C_VEL
LIN {X 0,Y 319.595,Z 467.908,A -85,B 0,C 180,E1 -15459.4,E2 -15459.4} C_VEL
LIN {X 0,Y 319.651,Z 467.917,A -85,B 0,C 180,E1 -15462.073,E2 -15462.073} C_VEL
LIN {X 0,Y 319.725,Z 467.907,A -85,B 0,C 180,E1 -15466.008,E2 -15466.008} C_VEL
LIN {X 0,Y 319.75,Z 467.891,A -85,B 0,C 180,E1 -15469.873,E2 -15469.873} C_VEL
LIN {X 0,Y 319.791,Z 467.892,A -85,B 0,C 180,E1 -15470.749,E2 -15470.749} C_VEL
LIN {X 0,Y 319.515,Z 467.935,A -85,B 0,C 180,E1 -15471.453,E2 -15471.453} C_VEL
LIN {X 0,Y 317.545,Z 468.193,A -85,B 0,C 180,E1 -15472.831,E2 -15472.831} C_VEL
LIN {X 0,Y 313.745,Z 468.665,A -85,B 0,C 180,E1 -15474.896,E2 -15474.896} C_VEL
LIN {X 0,Y 312.755,Z 468.778,A -85,B 0,C 180,E1 -15475.972,E2 -15475.972} C_VEL
LIN {X 0,Y 312.717,Z 468.777,A -85,B 0,C 180,E1 -15476.336,E2 -15476.336} C_VEL
LIN {X 0,Y 312.983,Z 468.726,A -85,B 0,C 180,E1 -15478.714,E2 -15478.714} C_VEL
LIN {X 0,Y 312.983,Z 468.751,A -85,B 0,C 180,E1 -15481.287,E2 -15481.287} C_VEL
LIN {X 0,Y 312.711,Z 468.775,A -85,B 0,C 180,E1 -15485.158,E2 -15485.158} C_VEL
LIN {X 0,Y 312.847,Z 468.746,A -85,B 0,C 180,E1 -15487.747,E2 -15487.747} C_VEL
LIN {X 0,Y 312.662,Z 468.781,A -85,B 0,C 180,E1 -15491.672,E2 -15491.672} C_VEL
LIN {X 0,Y 312.694,Z 468.778,A -85,B 0,C 180,E1 -15494.888,E2 -15494.888} C_VEL
LIN {X 0,Y 312.603,Z 468.725,A -85,B 0,C 180,E1 -15499.225,E2 -15499.225} C_VEL
LIN {X 0,Y 312.52,Z 468.773,A -85,B 0,C 180,E1 -15502.781,E2 -15502.781} C_VEL
LIN {X 0,Y 312.591,Z 468.767,A -85,B 0,C 180,E1 -15505.934,E2 -15505.934} C_VEL
LIN {X 0,Y 312.541,Z 468.75,A -85,B 0,C 180,E1 -15509.65,E2 -15509.65} C_VEL
LIN {X 0,Y 312.515,Z 468.777,A -85,B 0,C 180,E1 -15513.69,E2 -15513.69} C_VEL
LIN {X 0,Y 312.562,Z 468.836,A -85,B 0,C 180,E1 -15517.838,E2 -15517.838} C_VEL
LIN {X 0,Y 313.291,Z 471.122,A -85,B 0,C 180,E1 -15518.912,E2 -15518.912} C_VEL
LIN {X 0,Y 314.698,Z 475.35,A -85,B 0,C 180,E1 -15520.522,E2 -15520.522} C_VEL
LIN {X 0,Y 317.892,Z 480.352,A -85,B 0,C 180,E1 -15521.389,E2 -15521.389} C_VEL
LIN {X 0,Y 322.793,Z 488.093,A -85,B 0,C 180,E1 -15522.609,E2 -15522.609} C_VEL
LIN {X 0,Y 329.048,Z 498.418,A -85,B 0,C 180,E1 -15524.089,E2 -15524.089} C_VEL
LIN {X 0,Y 336.584,Z 511.72,A -85,B 0,C 180,E1 -15525.776,E2 -15525.776} C_VEL
LIN {X 0,Y 345.208,Z 528.674,A -85,B 0,C 180,E1 -15527.612,E2 -15527.612} C_VEL
LIN {X 0,Y 351.492,Z 542.326,A -85,B 0,C 180,E1 -15528.896,E2 -15528.896} C_VEL
LIN {X 0,Y 346.783,Z 660.904,A -85,B 0,C 180,E1 -15531.359,E2 -15531.359} C_VEL
LIN {X 0,Y 345.366,Z 691.023,A -85,B 0,C 180,E1 -15532.008,E2 -15532.008} C_VEL
LIN {X 0,Y 344.151,Z 705.48,A -85,B 0,C 180,E1 -15532.452,E2 -15532.452} C_VEL
LIN {X 0,Y 342.348,Z 720.922,A -85,B 0,C 180,E1 -15533.098,E2 -15533.098} C_VEL
LIN {X 0,Y 340.059,Z 736.921,A -85,B 0,C 180,E1 -15534.01,E2 -15534.01} C_VEL
LIN {X 0,Y 337.477,Z 751.561,A -85,B 0,C 180,E1 -15535.063,E2 -15535.063} C_VEL
LIN {X 0,Y 335.219,Z 763.202,A -85,B 0,C 180,E1 -15536.069,E2 -15536.069} C_VEL
LIN {X 0,Y 332.418,Z 776.03,A -85,B 0,C 180,E1 -15537.377,E2 -15537.377} C_VEL
LIN {X 0,Y 329.761,Z 787.442,A -85,B 0,C 180,E1 -15538.746,E2 -15538.746} C_VEL
LIN {X 0,Y 327.092,Z 798.005,A -85,B 0,C 180,E1 -15540.208,E2 -15540.208} C_VEL
LIN {X 0,Y 324.865,Z 806.689,A -85,B 0,C 180,E1 -15541.58,E2 -15541.58} C_VEL
LIN {X 0,Y 322.24,Z 816.734,A -85,B 0,C 180,E1 -15543.406,E2 -15543.406} C_VEL
LIN {X 0,Y 319.843,Z 825.859,A -85,B 0,C 180,E1 -15545.324,E2 -15545.324} C_VEL
LIN {X 0,Y 317.751,Z 833.751,A -85,B 0,C 180,E1 -15547.229,E2 -15547.229} C_VEL
LIN {X 0,Y 316.033,Z 840.718,A -85,B 0,C 180,E1 -15549.157,E2 -15549.157} C_VEL
LIN {X 0,Y 314.621,Z 846.862,A -85,B 0,C 180,E1 -15551.101,E2 -15551.101} C_VEL
LIN {X 0,Y 313.058,Z 853.81,A -85,B 0,C 180,E1 -15553.703,E2 -15553.703} C_VEL
LIN {X 0,Y 312.257,Z 858.284,A -85,B 0,C 180,E1 -15555.666,E2 -15555.666} C_VEL
LIN {X 0,Y 311.393,Z 863.184,A -85,B 0,C 180,E1 -15558.28,E2 -15558.28} C_VEL
LIN {X 0,Y 310.89,Z 867.035,A -85,B 0,C 180,E1 -15560.895,E2 -15560.895} C_VEL
LIN {X 0,Y 310.762,Z 869.889,A -85,B 0,C 180,E1 -15563.507,E2 -15563.507} C_VEL
LIN {X 0,Y 310.687,Z 871.773,A -85,B 0,C 180,E1 -15566.109,E2 -15566.109} C_VEL
LIN {X 0,Y 310.667,Z 872.448,A -85,B 0,C 180,E1 -15567.407,E2 -15567.407} C_VEL
LIN {X 0,Y 310.641,Z 872.92,A -85,B 0,C 180,E1 -15570,E2 -15570} C_VEL
LIN {X 0,Y 310.667,Z 872.448,A -85,B 0,C 180,E1 -15572.593,E2 -15572.593} C_VEL
LIN {X 0,Y 310.722,Z 870.654,A -85,B 0,C 180,E1 -15575.616,E2 -15575.616} C_VEL
LIN {X 0,Y 310.78,Z 868.637,A -85,B 0,C 180,E1 -15577.798,E2 -15577.798} C_VEL
LIN {X 0,Y 311.216,Z 864.223,A -85,B 0,C 180,E1 -15581.066,E2 -15581.066} C_VEL
LIN {X 0,Y 311.72,Z 860.855,A -85,B 0,C 180,E1 -15583.03,E2 -15583.03} C_VEL
LIN {X 0,Y 312.453,Z 856.871,A -85,B 0,C 180,E1 -15585.003,E2 -15585.003} C_VEL
LIN {X 0,Y 313.779,Z 850.495,A -85,B 0,C 180,E1 -15587.6,E2 -15587.6} C_VEL
LIN {X 0,Y 315.521,Z 842.825,A -85,B 0,C 180,E1 -15590.197,E2 -15590.197} C_VEL
LIN {X 0,Y 317.138,Z 836.17,A -85,B 0,C 180,E1 -15592.131,E2 -15592.131} C_VEL
LIN {X 0,Y 319.122,Z 828.617,A -85,B 0,C 180,E1 -15594.042,E2 -15594.042} C_VEL
LIN {X 0,Y 321.427,Z 820.033,A -85,B 0,C 180,E1 -15595.931,E2 -15595.931} C_VEL
LIN {X 0,Y 323.94,Z 810.241,A -85,B 0,C 180,E1 -15597.803,E2 -15597.803} C_VEL
LIN {X 0,Y 326.572,Z 800.018,A -85,B 0,C 180,E1 -15599.49,E2 -15599.49} C_VEL
LIN {X 0,Y 328.975,Z 790.596,A -85,B 0,C 180,E1 -15600.844,E2 -15600.844} C_VEL
LIN {X 0,Y 331.526,Z 779.946,A -85,B 0,C 180,E1 -15602.182,E2 -15602.182} C_VEL
LIN {X 0,Y 334.223,Z 767.7,A -85,B 0,C 180,E1 -15603.502,E2 -15603.502} C_VEL
LIN {X 0,Y 336.478,Z 756.785,A -85,B 0,C 180,E1 -15604.51,E2 -15604.51} C_VEL
LIN {X 0,Y 338.861,Z 744.055,A -85,B 0,C 180,E1 -15605.5,E2 -15605.5} C_VEL
LIN {X 0,Y 340.876,Z 731.265,A -85,B 0,C 180,E1 -15606.336,E2 -15606.336} C_VEL
LIN {X 0,Y 342.775,Z 717.386,A -85,B 0,C 180,E1 -15607.06,E2 -15607.06} C_VEL
LIN {X 0,Y 344.325,Z 703.777,A -85,B 0,C 180,E1 -15607.605,E2 -15607.605} C_VEL
LIN {X 0,Y 345.367,Z 691.023,A -85,B 0,C 180,E1 -15607.992,E2 -15607.992} C_VEL
LIN {X 0,Y 346.996,Z 653.737,A -85,B 0,C 180,E1 -15608.799,E2 -15608.799} C_VEL
LIN {X 0,Y 350.535,Z 567.16,A -85,B 0,C 180,E1 -15610.583,E2 -15610.583} C_VEL
LIN {X 0,Y 351.448,Z 542.242,A -85,B 0,C 180,E1 -15611.113,E2 -15611.113} C_VEL
LIN {X 0,Y 343.842,Z 525.845,A -85,B 0,C 180,E1 -15612.673,E2 -15612.673} C_VEL
LIN {X 0,Y 335.46,Z 509.66,A -85,B 0,C 180,E1 -15614.47,E2 -15614.47} C_VEL
LIN {X 0,Y 327.239,Z 495.289,A -85,B 0,C 180,E1 -15616.334,E2 -15616.334} C_VEL
LIN {X 0,Y 321.001,Z 485.269,A -85,B 0,C 180,E1 -15617.829,E2 -15617.829} C_VEL
LIN {X 0,Y 317.238,Z 479.544,A -85,B 0,C 180,E1 -15618.771,E2 -15618.771} C_VEL
LIN {X 0,Y 314.554,Z 475.033,A -85,B 0,C 180,E1 -15619.561,E2 -15619.561} C_VEL
LIN {X 0,Y 312.579,Z 469.01,A -85,B 0,C 180,E1 -15622.015,E2 -15622.015} C_VEL
LIN {X 0,Y 312.502,Z 468.772,A -85,B 0,C 180,E1 -15625.789,E2 -15625.789} C_VEL
LIN {X 0,Y 312.524,Z 468.789,A -85,B 0,C 180,E1 -15628.854,E2 -15628.854} C_VEL
LIN {X 0,Y 312.569,Z 468.736,A -85,B 0,C 180,E1 -15631.824,E2 -15631.824} C_VEL
LIN {X 0,Y 312.579,Z 468.788,A -85,B 0,C 180,E1 -15634.71,E2 -15634.71} C_VEL
LIN {X 0,Y 312.53,Z 468.735,A -85,B 0,C 180,E1 -15638.912,E2 -15638.912} C_VEL
LIN {X 0,Y 312.632,Z 468.734,A -85,B 0,C 180,E1 -15641.656,E2 -15641.656} C_VEL
LIN {X 0,Y 312.687,Z 468.77,A -85,B 0,C 180,E1 -15645.686,E2 -15645.686} C_VEL
LIN {X 0,Y 312.692,Z 468.781,A -85,B 0,C 180,E1 -15649.641,E2 -15649.641} C_VEL
LIN {X 0,Y 312.847,Z 468.747,A -85,B 0,C 180,E1 -15652.253,E2 -15652.253} C_VEL
LIN {X 0,Y 312.711,Z 468.776,A -85,B 0,C 180,E1 -15654.842,E2 -15654.842} C_VEL
LIN {X 0,Y 312.983,Z 468.749,A -85,B 0,C 180,E1 -15658.713,E2 -15658.713} C_VEL
LIN {X 0,Y 312.983,Z 468.724,A -85,B 0,C 180,E1 -15661.286,E2 -15661.286} C_VEL
LIN {X 0,Y 312.711,Z 468.766,A -85,B 0,C 180,E1 -15665.157,E2 -15665.157} C_VEL
LIN {X 0,Y 312.859,Z 468.751,A -85,B 0,C 180,E1 -15667.746,E2 -15667.746} C_VEL
LIN {X 0,Y 312.662,Z 468.767,A -85,B 0,C 180,E1 -15671.671,E2 -15671.671} C_VEL
LIN {X 0,Y 312.693,Z 468.769,A -85,B 0,C 180,E1 -15674.887,E2 -15674.887} C_VEL
LIN {X 0,Y 312.602,Z 468.787,A -85,B 0,C 180,E1 -15679.225,E2 -15679.225} C_VEL
LIN {X 0,Y 312.521,Z 468.807,A -85,B 0,C 180,E1 -15682.781,E2 -15682.781} C_VEL
LIN {X 0,Y 312.59,Z 468.734,A -85,B 0,C 180,E1 -15685.933,E2 -15685.933} C_VEL
LIN {X 0,Y 312.538,Z 468.791,A -85,B 0,C 180,E1 -15689.65,E2 -15689.65} C_VEL
LIN {X 0,Y 312.513,Z 468.751,A -85,B 0,C 180,E1 -15693.689,E2 -15693.689} C_VEL
LIN {X 0,Y 312.548,Z 468.805,A -85,B 0,C 180,E1 -15697.381,E2 -15697.381} C_VEL
LIN {X 0,Y 312.545,Z 468.945,A -85,B 0,C 180,E1 -15700.361,E2 -15700.361} C_VEL
LIN {X 0,Y 312.825,Z 470.108,A -85,B 0,C 180,E1 -15700.815,E2 -15700.815} C_VEL
LIN {X 0,Y 314.203,Z 472.569,A -85,B 0,C 180,E1 -15701.341,E2 -15701.341} C_VEL
LIN {X 0,Y 317.098,Z 474.856,A -85,B 0,C 180,E1 -15702.315,E2 -15702.315} C_VEL
LIN {X 0,Y 318.836,Z 477.771,A -85,B 0,C 180,E1 -15702.995,E2 -15702.995} C_VEL
LIN {X 0,Y 321.495,Z 480.009,A -85,B 0,C 180,E1 -15703.964,E2 -15703.964} C_VEL
LIN {X 0,Y 322.488,Z 481.041,A -85,B 0,C 180,E1 -15704.343,E2 -15704.343} C_VEL
LIN {X 0,Y 324.917,Z 484.303,A -85,B 0,C 180,E1 -15705.345,E2 -15705.345} C_VEL
LIN {X 0,Y 327.638,Z 486.539,A -85,B 0,C 180,E1 -15706.433,E2 -15706.433} C_VEL
LIN {X 0,Y 330.099,Z 489.871,A -85,B 0,C 180,E1 -15707.503,E2 -15707.503} C_VEL
LIN {X 0,Y 333.117,Z 492.464,A -85,B 0,C 180,E1 -15708.749,E2 -15708.749} C_VEL
LIN {X 0,Y 335.927,Z 495.97,A -85,B 0,C 180,E1 -15709.982,E2 -15709.982} C_VEL
LIN {X 0,Y 338.862,Z 498.407,A -85,B 0,C 180,E1 -15711.232,E2 -15711.232} C_VEL
LIN {X 0,Y 341.604,Z 501.832,A -85,B 0,C 180,E1 -15712.493,E2 -15712.493} C_VEL
LIN {X 0,Y 344.873,Z 504.572,A -85,B 0,C 180,E1 -15713.963,E2 -15713.963} C_VEL
LIN {X 0,Y 347.894,Z 508.176,A -85,B 0,C 180,E1 -15715.42,E2 -15715.42} C_VEL
LIN {X 0,Y 351.095,Z 510.804,A -85,B 0,C 180,E1 -15716.943,E2 -15716.943} C_VEL
LIN {X 0,Y 354.222,Z 514.423,A -85,B 0,C 180,E1 -15718.555,E2 -15718.555} C_VEL
LIN {X 0,Y 357.572,Z 517.034,A -85,B 0,C 180,E1 -15720.283,E2 -15720.283} C_VEL
LIN {X 0,Y 360.586,Z 520.554,A -85,B 0,C 180,E1 -15721.983,E2 -15721.983} C_VEL
LIN {X 0,Y 364.336,Z 523.523,A -85,B 0,C 180,E1 -15724.11,E2 -15724.11} C_VEL
LIN {X 0,Y 367.179,Z 526.964,A -85,B 0,C 180,E1 -15725.941,E2 -15725.941} C_VEL
LIN {X 0,Y 370.047,Z 529.051,A -85,B 0,C 180,E1 -15727.798,E2 -15727.798} C_VEL
LIN {X 0,Y 371.301,Z 529.925,A -85,B 0,C 180,E1 -15728.65,E2 -15728.65} C_VEL
LIN {X 0,Y 373.653,Z 532.887,A -85,B 0,C 180,E1 -15730.457,E2 -15730.457} C_VEL
LIN {X 0,Y 376.604,Z 535.199,A -85,B 0,C 180,E1 -15732.825,E2 -15732.825} C_VEL
LIN {X 0,Y 378.851,Z 536.555,A -85,B 0,C 180,E1 -15734.813,E2 -15734.813} C_VEL
LIN {X 0,Y 380.679,Z 539.174,A -85,B 0,C 180,E1 -15736.846,E2 -15736.846} C_VEL
LIN {X 0,Y 382.519,Z 540.915,A -85,B 0,C 180,E1 -15739.091,E2 -15739.091} C_VEL
LIN {X 0,Y 384.24,Z 541.838,A -85,B 0,C 180,E1 -15741.586,E2 -15741.586} C_VEL
LIN {X 0,Y 385.659,Z 542.585,A -85,B 0,C 180,E1 -15744.42,E2 -15744.42} C_VEL
LIN {X 0,Y 386.418,Z 543.037,A -85,B 0,C 180,E1 -15746.872,E2 -15746.872} C_VEL
LIN {X 0,Y 386.717,Z 543.257,A -85,B 0,C 180,E1 -15748.959,E2 -15748.959} C_VEL
LIN {X 0,Y 386.687,Z 543.182,A -85,B 0,C 180,E1 -15751.603,E2 -15751.603} C_VEL
LIN {X 0,Y 386.138,Z 542.947,A -85,B 0,C 180,E1 -15754.175,E2 -15754.175} C_VEL
LIN {X 0,Y 385.183,Z 542.325,A -85,B 0,C 180,E1 -15756.676,E2 -15756.676} C_VEL
LIN {X 0,Y 383.54,Z 541.546,A -85,B 0,C 180,E1 -15759.492,E2 -15759.492} C_VEL
LIN {X 0,Y 381.492,Z 540.034,A -85,B 0,C 180,E1 -15762.224,E2 -15762.224} C_VEL
LIN {X 0,Y 379.486,Z 537.61,A -85,B 0,C 180,E1 -15764.491,E2 -15764.491} C_VEL
LIN {X 0,Y 378.587,Z 536.245,A -85,B 0,C 180,E1 -15765.438,E2 -15765.438} C_VEL
LIN {X 0,Y 375.624,Z 534.572,A -85,B 0,C 180,E1 -15767.983,E2 -15767.983} C_VEL
LIN {X 0,Y 372.978,Z 532.171,A -85,B 0,C 180,E1 -15770.073,E2 -15770.073} C_VEL
LIN {X 0,Y 371.131,Z 529.58,A -85,B 0,C 180,E1 -15771.493,E2 -15771.493} C_VEL
LIN {X 0,Y 367.804,Z 527.552,A -85,B 0,C 180,E1 -15773.657,E2 -15773.657} C_VEL
LIN {X 0,Y 364.839,Z 524.304,A -85,B 0,C 180,E1 -15775.557,E2 -15775.557} C_VEL
LIN {X 0,Y 363.732,Z 522.853,A -85,B 0,C 180,E1 -15776.253,E2 -15776.253} C_VEL
LIN {X 0,Y 360.188,Z 520.207,A -85,B 0,C 180,E1 -15778.242,E2 -15778.242} C_VEL
LIN {X 0,Y 357.064,Z 516.486,A -85,B 0,C 180,E1 -15780,E2 -15780} C_VEL
LIN {X 0,Y 353.673,Z 513.883,A -85,B 0,C 180,E1 -15781.727,E2 -15781.727} C_VEL
LIN {X 0,Y 350.262,Z 510.035,A -85,B 0,C 180,E1 -15783.45,E2 -15783.45} C_VEL
LIN {X 0,Y 346.743,Z 507.045,A -85,B 0,C 180,E1 -15785.115,E2 -15785.115} C_VEL
LIN {X 0,Y 344.163,Z 503.844,A -85,B 0,C 180,E1 -15786.358,E2 -15786.358} C_VEL
LIN {X 0,Y 340.822,Z 501.051,A -85,B 0,C 180,E1 -15787.849,E2 -15787.849} C_VEL
LIN {X 0,Y 338.219,Z 497.757,A -85,B 0,C 180,E1 -15789.048,E2 -15789.048} C_VEL
LIN {X 0,Y 335.134,Z 495.1,A -85,B 0,C 180,E1 -15790.371,E2 -15790.371} C_VEL
LIN {X 0,Y 332.752,Z 492.007,A -85,B 0,C 180,E1 -15791.413,E2 -15791.413} C_VEL
LIN {X 0,Y 329.484,Z 489.181,A -85,B 0,C 180,E1 -15792.757,E2 -15792.757} C_VEL
LIN {X 0,Y 327.237,Z 486.077,A -85,B 0,C 180,E1 -15793.73,E2 -15793.73} C_VEL
LIN {X 0,Y 324.417,Z 483.768,A -85,B 0,C 180,E1 -15794.86,E2 -15794.86} C_VEL
LIN {X 0,Y 321.735,Z 480.156,A -85,B 0,C 180,E1 -15795.951,E2 -15795.951} C_VEL
LIN {X 0,Y 319.04,Z 477.998,A -85,B 0,C 180,E1 -15796.931,E2 -15796.931} C_VEL
LIN {X 0,Y 317.092,Z 474.919,A -85,B 0,C 180,E1 -15797.684,E2 -15797.684} C_VEL
LIN {X 0,Y 313.889,Z 472.186,A -85,B 0,C 180,E1 -15798.769,E2 -15798.769} C_VEL
LIN {X 0,Y 312.664,Z 469.631,A -85,B 0,C 180,E1 -15799.319,E2 -15799.319} C_VEL
LIN {X 0,Y 312.555,Z 468.847,A -85,B 0,C 180,E1 -15799.809,E2 -15799.809} C_VEL
LIN {X 0,Y 312.548,Z 468.805,A -85,B 0,C 180,E1 -15802.619,E2 -15802.619} C_VEL
LIN {X 0,Y 312.513,Z 468.751,A -85,B 0,C 180,E1 -15806.311,E2 -15806.311} C_VEL
LIN {X 0,Y 312.538,Z 468.791,A -85,B 0,C 180,E1 -15810.35,E2 -15810.35} C_VEL
LIN {X 0,Y 312.59,Z 468.734,A -85,B 0,C 180,E1 -15814.067,E2 -15814.067} C_VEL
LIN {X 0,Y 312.559,Z 468.802,A -85,B 0,C 180,E1 -15817.527,E2 -15817.527} C_VEL
LIN {X 0,Y 312.631,Z 468.794,A -85,B 0,C 180,E1 -15821.656,E2 -15821.656} C_VEL
LIN {X 0,Y 312.686,Z 468.778,A -85,B 0,C 180,E1 -15825.686,E2 -15825.686} C_VEL
LIN {X 0,Y 312.694,Z 468.766,A -85,B 0,C 180,E1 -15829.642,E2 -15829.642} C_VEL
LIN {X 0,Y 312.859,Z 468.753,A -85,B 0,C 180,E1 -15832.254,E2 -15832.254} C_VEL
LIN {X 0,Y 312.711,Z 468.769,A -85,B 0,C 180,E1 -15834.843,E2 -15834.843} C_VEL
LIN {X 0,Y 312.717,Z 468.777,A -85,B 0,C 180,E1 -15836.336,E2 -15836.336} C_VEL
LIN {X 0,Y 312.185,Z 468.835,A -85,B 0,C 180,E1 -15837.414,E2 -15837.414} C_VEL
LIN {X 0,Y 309.45,Z 469.179,A -85,B 0,C 180,E1 -15839.171,E2 -15839.171} C_VEL
LIN {X 0,Y 307.045,Z 469.487,A -85,B 0,C 180,E1 -15840.596,E2 -15840.596} C_VEL
LIN {X 0,Y 305.986,Z 469.617,A -85,B 0,C 180,E1 -15841.698,E2 -15841.698} C_VEL
LIN {X 0,Y 305.89,Z 469.622,A -85,B 0,C 180,E1 -15842.072,E2 -15842.072} C_VEL
LIN {X 0,Y 305.837,Z 469.636,A -85,B 0,C 180,E1 -15846.598,E2 -15846.598} C_VEL
LIN {X 0,Y 305.697,Z 469.635,A -85,B 0,C 180,E1 -15849.261,E2 -15849.261} C_VEL
LIN {X 0,Y 305.581,Z 469.649,A -85,B 0,C 180,E1 -15853.297,E2 -15853.297} C_VEL
LIN {X 0,Y 305.587,Z 469.666,A -85,B 0,C 180,E1 -15856.021,E2 -15856.021} C_VEL
LIN {X 0,Y 305.554,Z 469.599,A -85,B 0,C 180,E1 -15859.436,E2 -15859.436} C_VEL
LIN {X 0,Y 305.481,Z 469.656,A -85,B 0,C 180,E1 -15863.04,E2 -15863.04} C_VEL
LIN {X 0,Y 305.521,Z 469.638,A -85,B 0,C 180,E1 -15866.219,E2 -15866.219} C_VEL
LIN {X 0,Y 305.49,Z 469.62,A -85,B 0,C 180,E1 -15869.05,E2 -15869.05} C_VEL
LIN {X 0,Y 305.473,Z 469.686,A -85,B 0,C 180,E1 -15871.949,E2 -15871.949} C_VEL
LIN {X 0,Y 305.458,Z 469.646,A -85,B 0,C 180,E1 -15875.114,E2 -15875.114} C_VEL
LIN {X 0,Y 305.514,Z 469.875,A -85,B 0,C 180,E1 -15876.734,E2 -15876.734} C_VEL
LIN {X 0,Y 307.192,Z 474.715,A -85,B 0,C 180,E1 -15878.814,E2 -15878.814} C_VEL
LIN {X 0,Y 309.913,Z 479.276,A -85,B 0,C 180,E1 -15879.661,E2 -15879.661} C_VEL
LIN {X 0,Y 311.747,Z 481.847,A -85,B 0,C 180,E1 -15880.153,E2 -15880.153} C_VEL
LIN {X 0,Y 316.114,Z 488.575,A -85,B 0,C 180,E1 -15881.302,E2 -15881.302} C_VEL
LIN {X 0,Y 321.776,Z 497.703,A -85,B 0,C 180,E1 -15882.722,E2 -15882.722} C_VEL
LIN {X 0,Y 330.089,Z 512.118,A -85,B 0,C 180,E1 -15884.689,E2 -15884.689} C_VEL
LIN {X 0,Y 337.242,Z 525.864,A -85,B 0,C 180,E1 -15886.292,E2 -15886.292} C_VEL
LIN {X 0,Y 345.048,Z 542.379,A -85,B 0,C 180,E1 -15887.964,E2 -15887.964} C_VEL
LIN {X 0,Y 346.115,Z 544.817,A -85,B 0,C 180,E1 -15888.188,E2 -15888.188} C_VEL
LIN {X 0,Y 340.405,Z 680.395,A -85,B 0,C 180,E1 -15891.02,E2 -15891.02} C_VEL
LIN {X 0,Y 339.114,Z 699.269,A -85,B 0,C 180,E1 -15891.511,E2 -15891.511} C_VEL
LIN {X 0,Y 337.553,Z 713.803,A -85,B 0,C 180,E1 -15892.06,E2 -15892.06} C_VEL
LIN {X 0,Y 335.757,Z 727.128,A -85,B 0,C 180,E1 -15892.72,E2 -15892.72} C_VEL
LIN {X 0,Y 333.639,Z 740.518,A -85,B 0,C 180,E1 -15893.554,E2 -15893.554} C_VEL
LIN {X 0,Y 331.302,Z 753.091,A -85,B 0,C 180,E1 -15894.5,E2 -15894.5} C_VEL
LIN {X 0,Y 328.968,Z 764.49,A -85,B 0,C 180,E1 -15895.519,E2 -15895.519} C_VEL
LIN {X 0,Y 326.399,Z 775.818,A -85,B 0,C 180,E1 -15896.698,E2 -15896.698} C_VEL
LIN {X 0,Y 324.032,Z 785.666,A -85,B 0,C 180,E1 -15897.879,E2 -15897.879} C_VEL
LIN {X 0,Y 321.204,Z 796.788,A -85,B 0,C 180,E1 -15899.423,E2 -15899.423} C_VEL
LIN {X 0,Y 318.539,Z 806.476,A -85,B 0,C 180,E1 -15900.963,E2 -15900.963} C_VEL
LIN {X 0,Y 315.886,Z 816.21,A -85,B 0,C 180,E1 -15902.757,E2 -15902.757} C_VEL
LIN {X 0,Y 313.332,Z 825.647,A -85,B 0,C 180,E1 -15904.776,E2 -15904.776} C_VEL
LIN {X 0,Y 311.118,Z 833.538,A -85,B 0,C 180,E1 -15906.715,E2 -15906.715} C_VEL
LIN {X 0,Y 309.255,Z 840.596,A -85,B 0,C 180,E1 -15908.709,E2 -15908.709} C_VEL
LIN {X 0,Y 307.804,Z 846.649,A -85,B 0,C 180,E1 -15910.666,E2 -15910.666} C_VEL
LIN {X 0,Y 306.133,Z 853.597,A -85,B 0,C 180,E1 -15913.324,E2 -15913.324} C_VEL
LIN {X 0,Y 305.283,Z 858.071,A -85,B 0,C 180,E1 -15915.331,E2 -15915.331} C_VEL
LIN {X 0,Y 304.357,Z 862.971,A -85,B 0,C 180,E1 -15918.006,E2 -15918.006} C_VEL
LIN {X 0,Y 303.833,Z 866.824,A -85,B 0,C 180,E1 -15920.682,E2 -15920.682} C_VEL
LIN {X 0,Y 303.678,Z 869.678,A -85,B 0,C 180,E1 -15923.355,E2 -15923.355} C_VEL
LIN {X 0,Y 303.602,Z 871.563,A -85,B 0,C 180,E1 -15926.018,E2 -15926.018} C_VEL
LIN {X 0,Y 303.592,Z 872.239,A -85,B 0,C 180,E1 -15927.346,E2 -15927.346} C_VEL
LIN {X 0,Y 303.556,Z 872.711,A -85,B 0,C 180,E1 -15930,E2 -15930} C_VEL
LIN {X 0,Y 303.591,Z 872.239,A -85,B 0,C 180,E1 -15932.654,E2 -15932.654} C_VEL
LIN {X 0,Y 303.624,Z 870.617,A -85,B 0,C 180,E1 -15935.544,E2 -15935.544} C_VEL
LIN {X 0,Y 303.69,Z 868.426,A -85,B 0,C 180,E1 -15937.981,E2 -15937.981} C_VEL
LIN {X 0,Y 304.172,Z 864.011,A -85,B 0,C 180,E1 -15941.326,E2 -15941.326} C_VEL
LIN {X 0,Y 304.731,Z 860.643,A -85,B 0,C 180,E1 -15943.334,E2 -15943.334} C_VEL
LIN {X 0,Y 305.8,Z 855.142,A -85,B 0,C 180,E1 -15946.009,E2 -15946.009} C_VEL
LIN {X 0,Y 306.921,Z 850.283,A -85,B 0,C 180,E1 -15948.006,E2 -15948.006} C_VEL
LIN {X 0,Y 308.769,Z 842.612,A -85,B 0,C 180,E1 -15950.658,E2 -15950.658} C_VEL
LIN {X 0,Y 310.471,Z 835.957,A -85,B 0,C 180,E1 -15952.632,E2 -15952.632} C_VEL
LIN {X 0,Y 312.526,Z 828.404,A -85,B 0,C 180,E1 -15954.583,E2 -15954.583} C_VEL
LIN {X 0,Y 314.937,Z 819.82,A -85,B 0,C 180,E1 -15956.507,E2 -15956.507} C_VEL
LIN {X 0,Y 317.586,Z 810.028,A -85,B 0,C 180,E1 -15958.41,E2 -15958.41} C_VEL
LIN {X 0,Y 320.34,Z 799.805,A -85,B 0,C 180,E1 -15960.122,E2 -15960.122} C_VEL
LIN {X 0,Y 323.142,Z 789.085,A -85,B 0,C 180,E1 -15961.672,E2 -15961.672} C_VEL
LIN {X 0,Y 325.779,Z 778.429,A -85,B 0,C 180,E1 -15963.004,E2 -15963.004} C_VEL
LIN {X 0,Y 328.284,Z 767.489,A -85,B 0,C 180,E1 -15964.191,E2 -15964.191} C_VEL
LIN {X 0,Y 330.601,Z 756.574,A -85,B 0,C 180,E1 -15965.213,E2 -15965.213} C_VEL
LIN {X 0,Y 333.077,Z 743.844,A -85,B 0,C 180,E1 -15966.213,E2 -15966.213} C_VEL
LIN {X 0,Y 335.203,Z 730.785,A -85,B 0,C 180,E1 -15967.073,E2 -15967.073} C_VEL
LIN {X 0,Y 337.069,Z 717.634,A -85,B 0,C 180,E1 -15967.768,E2 -15967.768} C_VEL
LIN {X 0,Y 338.662,Z 704.266,A -85,B 0,C 180,E1 -15968.313,E2 -15968.313} C_VEL
LIN {X 0,Y 339.785,Z 690.813,A -85,B 0,C 180,E1 -15968.731,E2 -15968.731} C_VEL
LIN {X 0,Y 341.419,Z 655.318,A -85,B 0,C 180,E1 -15969.508,E2 -15969.508} C_VEL
LIN {X 0,Y 345.171,Z 566.799,A -85,B 0,C 180,E1 -15971.354,E2 -15971.354} C_VEL
LIN {X 0,Y 346.092,Z 544.738,A -85,B 0,C 180,E1 -15971.818,E2 -15971.818} C_VEL
LIN {X 0,Y 337.927,Z 527.196,A -85,B 0,C 180,E1 -15973.56,E2 -15973.56} C_VEL
LIN {X 0,Y 330.852,Z 513.662,A -85,B 0,C 180,E1 -15975.133,E2 -15975.133} C_VEL
LIN {X 0,Y 323.05,Z 499.8,A -85,B 0,C 180,E1 -15976.969,E2 -15976.969} C_VEL
LIN {X 0,Y 317.392,Z 490.558,A -85,B 0,C 180,E1 -15978.372,E2 -15978.372} C_VEL
LIN {X 0,Y 313.324,Z 484.384,A -85,B 0,C 180,E1 -15979.422,E2 -15979.422} C_VEL
LIN {X 0,Y 310.299,Z 479.773,A -85,B 0,C 180,E1 -15980.236,E2 -15980.236} C_VEL
LIN {X 0,Y 307.897,Z 476.241,A -85,B 0,C 180,E1 -15980.901,E2 -15980.901} C_VEL
LIN {X 0,Y 307.116,Z 474.446,A -85,B 0,C 180,E1 -15981.27,E2 -15981.27} C_VEL
LIN {X 0,Y 305.503,Z 469.769,A -85,B 0,C 180,E1 -15983.385,E2 -15983.385} C_VEL
LIN {X 0,Y 305.461,Z 469.657,A -85,B 0,C 180,E1 -15986.483,E2 -15986.483} C_VEL
LIN {X 0,Y 305.46,Z 469.645,A -85,B 0,C 180,E1 -15989.591,E2 -15989.591} C_VEL
LIN {X 0,Y 305.494,Z 469.621,A -85,B 0,C 180,E1 -15992.606,E2 -15992.606} C_VEL
LIN {X 0,Y 305.499,Z 469.681,A -85,B 0,C 180,E1 -15995.538,E2 -15995.538} C_VEL
LIN {X 0,Y 305.5,Z 469.603,A -85,B 0,C 180,E1 -15999.814,E2 -15999.814} C_VEL
LIN {X 0,Y 305.568,Z 469.636,A -85,B 0,C 180,E1 -16002.602,E2 -16002.602} C_VEL
LIN {X 0,Y 305.642,Z 469.651,A -85,B 0,C 180,E1 -16005.348,E2 -16005.348} C_VEL
LIN {X 0,Y 305.629,Z 469.663,A -85,B 0,C 180,E1 -16009.399,E2 -16009.399} C_VEL
LIN {X 0,Y 305.791,Z 469.624,A -85,B 0,C 180,E1 -16012.074,E2 -16012.074} C_VEL
LIN {X 0,Y 305.682,Z 469.653,A -85,B 0,C 180,E1 -16014.723,E2 -16014.723} C_VEL
LIN {X 0,Y 305.95,Z 469.625,A -85,B 0,C 180,E1 -16018.683,E2 -16018.683} C_VEL
LIN {X 0,Y 305.95,Z 469.599,A -85,B 0,C 180,E1 -16021.316,E2 -16021.316} C_VEL
LIN {X 0,Y 305.682,Z 469.64,A -85,B 0,C 180,E1 -16025.276,E2 -16025.276} C_VEL
LIN {X 0,Y 305.802,Z 469.632,A -85,B 0,C 180,E1 -16027.926,E2 -16027.926} C_VEL
LIN {X 0,Y 305.596,Z 469.649,A -85,B 0,C 180,E1 -16031.945,E2 -16031.945} C_VEL
LIN {X 0,Y 305.631,Z 469.647,A -85,B 0,C 180,E1 -16035.034,E2 -16035.034} C_VEL
LIN {X 0,Y 305.573,Z 469.668,A -85,B 0,C 180,E1 -16038.783,E2 -16038.783} C_VEL
LIN {X 0,Y 305.479,Z 469.681,A -85,B 0,C 180,E1 -16043.039,E2 -16043.039} C_VEL
LIN {X 0,Y 305.519,Z 469.611,A -85,B 0,C 180,E1 -16046.219,E2 -16046.219} C_VEL
LIN {X 0,Y 305.488,Z 469.647,A -85,B 0,C 180,E1 -16049.05,E2 -16049.05} C_VEL
LIN {X 0,Y 305.437,Z 469.656,A -85,B 0,C 180,E1 -16051.952,E2 -16051.952} C_VEL
LIN {X 0,Y 305.456,Z 469.635,A -85,B 0,C 180,E1 -16055.113,E2 -16055.113} C_VEL
LIN {X 0,Y 305.531,Z 469.95,A -85,B 0,C 180,E1 -16058.55,E2 -16058.55} C_VEL
LIN {X 0,Y 305.865,Z 471.178,A -85,B 0,C 180,E1 -16058.944,E2 -16058.944} C_VEL
LIN {X 0,Y 307.343,Z 473.647,A -85,B 0,C 180,E1 -16059.446,E2 -16059.446} C_VEL
LIN {X 0,Y 309.711,Z 475.549,A -85,B 0,C 180,E1 -16060.181,E2 -16060.181} C_VEL
LIN {X 0,Y 311.603,Z 478.596,A -85,B 0,C 180,E1 -16060.849,E2 -16060.849} C_VEL
LIN {X 0,Y 314.742,Z 481.444,A -85,B 0,C 180,E1 -16061.897,E2 -16061.897} C_VEL
LIN {X 0,Y 317.02,Z 484.57,A -85,B 0,C 180,E1 -16062.732,E2 -16062.732} C_VEL
LIN {X 0,Y 320.133,Z 487.166,A -85,B 0,C 180,E1 -16063.849,E2 -16063.849} C_VEL
LIN {X 0,Y 322.651,Z 490.459,A -85,B 0,C 180,E1 -16064.853,E2 -16064.853} C_VEL
LIN {X 0,Y 325.725,Z 493.207,A -85,B 0,C 180,E1 -16066.079,E2 -16066.079} C_VEL
LIN {X 0,Y 328.54,Z 496.691,A -85,B 0,C 180,E1 -16067.269,E2 -16067.269} C_VEL
LIN {X 0,Y 331.436,Z 499.262,A -85,B 0,C 180,E1 -16068.456,E2 -16068.456} C_VEL
LIN {X 0,Y 334.459,Z 502.825,A -85,B 0,C 180,E1 -16069.767,E2 -16069.767} C_VEL
LIN {X 0,Y 337.173,Z 505.173,A -85,B 0,C 180,E1 -16070.934,E2 -16070.934} C_VEL
LIN {X 0,Y 340.139,Z 508.683,A -85,B 0,C 180,E1 -16072.282,E2 -16072.282} C_VEL
LIN {X 0,Y 343.225,Z 511.299,A -85,B 0,C 180,E1 -16073.663,E2 -16073.663} C_VEL
LIN {X 0,Y 346.294,Z 514.846,A -85,B 0,C 180,E1 -16075.126,E2 -16075.126} C_VEL
LIN {X 0,Y 349.557,Z 517.575,A -85,B 0,C 180,E1 -16076.671,E2 -16076.671} C_VEL
LIN {X 0,Y 352.774,Z 521.168,A -85,B 0,C 180,E1 -16078.297,E2 -16078.297} C_VEL
LIN {X 0,Y 356.194,Z 523.87,A -85,B 0,C 180,E1 -16080.042,E2 -16080.042} C_VEL
LIN {X 0,Y 359.333,Z 527.444,A -85,B 0,C 180,E1 -16081.798,E2 -16081.798} C_VEL
LIN {X 0,Y 362.937,Z 530.244,A -85,B 0,C 180,E1 -16083.828,E2 -16083.828} C_VEL
LIN {X 0,Y 365.832,Z 533.704,A -85,B 0,C 180,E1 -16085.653,E2 -16085.653} C_VEL
LIN {X 0,Y 368.845,Z 535.943,A -85,B 0,C 180,E1 -16087.6,E2 -16087.6} C_VEL
LIN {X 0,Y 370.171,Z 536.879,A -85,B 0,C 180,E1 -16088.481,E2 -16088.481} C_VEL
LIN {X 0,Y 372.587,Z 539.834,A -85,B 0,C 180,E1 -16090.326,E2 -16090.326} C_VEL
LIN {X 0,Y 375.518,Z 542.143,A -85,B 0,C 180,E1 -16092.645,E2 -16092.645} C_VEL
LIN {X 0,Y 377.778,Z 543.513,A -85,B 0,C 180,E1 -16094.642,E2 -16094.642} C_VEL
LIN {X 0,Y 379.686,Z 546.148,A -85,B 0,C 180,E1 -16096.712,E2 -16096.712} C_VEL
LIN {X 0,Y 381.622,Z 547.963,A -85,B 0,C 180,E1 -16099.065,E2 -16099.065} C_VEL
LIN {X 0,Y 383.475,Z 548.959,A -85,B 0,C 180,E1 -16101.752,E2 -16101.752} C_VEL
LIN {X 0,Y 384.784,Z 549.633,A -85,B 0,C 180,E1 -16104.407,E2 -16104.407} C_VEL
LIN {X 0,Y 385.551,Z 550.083,A -85,B 0,C 180,E1 -16106.865,E2 -16106.865} C_VEL
LIN {X 0,Y 385.851,Z 550.303,A -85,B 0,C 180,E1 -16108.956,E2 -16108.956} C_VEL
LIN {X 0,Y 385.851,Z 550.306,A -85,B 0,C 180,E1 -16111.044,E2 -16111.044} C_VEL
LIN {X 0,Y 385.552,Z 550.083,A -85,B 0,C 180,E1 -16113.135,E2 -16113.135} C_VEL
LIN {X 0,Y 384.787,Z 549.605,A -85,B 0,C 180,E1 -16115.591,E2 -16115.591} C_VEL
LIN {X 0,Y 383.353,Z 548.917,A -85,B 0,C 180,E1 -16118.433,E2 -16118.433} C_VEL
LIN {X 0,Y 381.452,Z 547.804,A -85,B 0,C 180,E1 -16121.152,E2 -16121.152} C_VEL
LIN {X 0,Y 379.665,Z 546.07,A -85,B 0,C 180,E1 -16123.32,E2 -16123.32} C_VEL
LIN {X 0,Y 377.535,Z 543.214,A -85,B 0,C 180,E1 -16125.595,E2 -16125.595} C_VEL
LIN {X 0,Y 374.479,Z 541.476,A -85,B 0,C 180,E1 -16128.184,E2 -16128.184} C_VEL
LIN {X 0,Y 371.737,Z 538.904,A -85,B 0,C 180,E1 -16130.349,E2 -16130.349} C_VEL
LIN {X 0,Y 369.931,Z 536.492,A -85,B 0,C 180,E1 -16131.713,E2 -16131.713} C_VEL
LIN {X 0,Y 366.4,Z 534.246,A -85,B 0,C 180,E1 -16133.976,E2 -16133.976} C_VEL
LIN {X 0,Y 363.371,Z 530.888,A -85,B 0,C 180,E1 -16135.907,E2 -16135.907} C_VEL
LIN {X 0,Y 362.247,Z 529.605,A -85,B 0,C 180,E1 -16136.572,E2 -16136.572} C_VEL
LIN {X 0,Y 358.851,Z 527.022,A -85,B 0,C 180,E1 -16138.476,E2 -16138.476} C_VEL
LIN {X 0,Y 355.704,Z 523.31,A -85,B 0,C 180,E1 -16140.228,E2 -16140.228} C_VEL
LIN {X 0,Y 352.172,Z 520.625,A -85,B 0,C 180,E1 -16141.996,E2 -16141.996} C_VEL
LIN {X 0,Y 348.727,Z 516.769,A -85,B 0,C 180,E1 -16143.728,E2 -16143.728} C_VEL
LIN {X 0,Y 345.08,Z 513.648,A -85,B 0,C 180,E1 -16145.448,E2 -16145.448} C_VEL
LIN {X 0,Y 342.607,Z 510.606,A -85,B 0,C 180,E1 -16146.623,E2 -16146.623} C_VEL
LIN {X 0,Y 339.001,Z 507.542,A -85,B 0,C 180,E1 -16148.224,E2 -16148.224} C_VEL
LIN {X 0,Y 336.437,Z 504.363,A -85,B 0,C 180,E1 -16149.385,E2 -16149.385} C_VEL
LIN {X 0,Y 333.301,Z 501.661,A -85,B 0,C 180,E1 -16150.718,E2 -16150.718} C_VEL
LIN {X 0,Y 330.821,Z 498.538,A -85,B 0,C 180,E1 -16151.812,E2 -16151.812} C_VEL
LIN {X 0,Y 327.357,Z 495.393,A -85,B 0,C 180,E1 -16153.237,E2 -16153.237} C_VEL
LIN {X 0,Y 325.12,Z 492.55,A -85,B 0,C 180,E1 -16154.171,E2 -16154.171} C_VEL
LIN {X 0,Y 321.934,Z 489.689,A -85,B 0,C 180,E1 -16155.432,E2 -16155.432} C_VEL
LIN {X 0,Y 319.775,Z 486.751,A -85,B 0,C 180,E1 -16156.288,E2 -16156.288} C_VEL
LIN {X 0,Y 316.767,Z 484.287,A -85,B 0,C 180,E1 -16157.361,E2 -16157.361} C_VEL
LIN {X 0,Y 314.23,Z 480.796,A -85,B 0,C 180,E1 -16158.286,E2 -16158.286} C_VEL
LIN {X 0,Y 311.439,Z 478.419,A -85,B 0,C 180,E1 -16159.206,E2 -16159.206} C_VEL
LIN {X 0,Y 309.373,Z 475.163,A -85,B 0,C 180,E1 -16159.927,E2 -16159.927} C_VEL
LIN {X 0,Y 307.01,Z 473.261,A -85,B 0,C 180,E1 -16160.659,E2 -16160.659} C_VEL
LIN {X 0,Y 305.623,Z 470.405,A -85,B 0,C 180,E1 -16161.247,E2 -16161.247} C_VEL
LIN {X 0,Y 305.516,Z 469.751,A -85,B 0,C 180,E1 -16161.604,E2 -16161.604} C_VEL
LIN {X 0,Y 305.456,Z 469.635,A -85,B 0,C 180,E1 -16164.887,E2 -16164.887} C_VEL
LIN {X 0,Y 305.445,Z 469.663,A -85,B 0,C 180,E1 -16168.355,E2 -16168.355} C_VEL
LIN {X 0,Y 305.513,Z 469.64,A -85,B 0,C 180,E1 -16171.114,E2 -16171.114} C_VEL
LIN {X 0,Y 305.558,Z 469.609,A -85,B 0,C 180,E1 -16174.087,E2 -16174.087} C_VEL
LIN {X 0,Y 305.475,Z 469.674,A -85,B 0,C 180,E1 -16178.401,E2 -16178.401} C_VEL
LIN {X 0,Y 305.573,Z 469.667,A -85,B 0,C 180,E1 -16181.217,E2 -16181.217} C_VEL
LIN {X 0,Y 305.642,Z 469.65,A -85,B 0,C 180,E1 -16185.349,E2 -16185.349} C_VEL
LIN {X 0,Y 305.63,Z 469.643,A -85,B 0,C 180,E1 -16189.4,E2 -16189.4} C_VEL
LIN {X 0,Y 305.802,Z 469.634,A -85,B 0,C 180,E1 -16192.074,E2 -16192.074} C_VEL
LIN {X 0,Y 305.682,Z 469.642,A -85,B 0,C 180,E1 -16194.724,E2 -16194.724} C_VEL
LIN {X 0,Y 305.95,Z 469.602,A -85,B 0,C 180,E1 -16198.684,E2 -16198.684} C_VEL
LIN {X 0,Y 305.95,Z 469.626,A -85,B 0,C 180,E1 -16201.317,E2 -16201.317} C_VEL
LIN {X 0,Y 305.89,Z 469.622,A -85,B 0,C 180,E1 -16202.072,E2 -16202.072} C_VEL
LIN {X 0,Y 305.184,Z 469.704,A -85,B 0,C 180,E1 -16203.169,E2 -16203.169} C_VEL
LIN {X 0,Y 302.282,Z 470.07,A -85,B 0,C 180,E1 -16204.954,E2 -16204.954} C_VEL
LIN {X 0,Y 299.844,Z 470.383,A -85,B 0,C 180,E1 -16206.402,E2 -16206.402} C_VEL
LIN {X 0,Y 298.81,Z 470.497,A -85,B 0,C 180,E1 -16207.525,E2 -16207.525} C_VEL
LIN {X 0,Y 298.731,Z 470.502,A -85,B 0,C 180,E1 -16207.905,E2 -16207.905} C_VEL
LIN {X 0,Y 298.546,Z 470.531,A -85,B 0,C 180,E1 -16212.232,E2 -16212.232} C_VEL
LIN {X 0,Y 298.579,Z 470.539,A -85,B 0,C 180,E1 -16215.195,E2 -16215.195} C_VEL
LIN {X 0,Y 298.519,Z 470.475,A -85,B 0,C 180,E1 -16219.245,E2 -16219.245} C_VEL
LIN {X 0,Y 298.45,Z 470.547,A -85,B 0,C 180,E1 -16223.598,E2 -16223.598} C_VEL
LIN {X 0,Y 298.479,Z 470.506,A -85,B 0,C 180,E1 -16226.576,E2 -16226.576} C_VEL
LIN {X 0,Y 298.417,Z 470.506,A -85,B 0,C 180,E1 -16229.642,E2 -16229.642} C_VEL
LIN {X 0,Y 298.404,Z 470.549,A -85,B 0,C 180,E1 -16232.799,E2 -16232.799} C_VEL
LIN {X 0,Y 298.455,Z 470.667,A -85,B 0,C 180,E1 -16235.337,E2 -16235.337} C_VEL
LIN {X 0,Y 299.748,Z 474.499,A -85,B 0,C 180,E1 -16237.038,E2 -16237.038} C_VEL
LIN {X 0,Y 302.907,Z 479.254,A -85,B 0,C 180,E1 -16238.046,E2 -16238.046} C_VEL
LIN {X 0,Y 304.343,Z 481.372,A -85,B 0,C 180,E1 -16238.466,E2 -16238.466} C_VEL
LIN {X 0,Y 308.593,Z 487.757,A -85,B 0,C 180,E1 -16239.669,E2 -16239.669} C_VEL
LIN {X 0,Y 313.205,Z 494.941,A -85,B 0,C 180,E1 -16240.915,E2 -16240.915} C_VEL
LIN {X 0,Y 320.615,Z 507.254,A -85,B 0,C 180,E1 -16242.807,E2 -16242.807} C_VEL
LIN {X 0,Y 328.422,Z 521.461,A -85,B 0,C 180,E1 -16244.68,E2 -16244.68} C_VEL
LIN {X 0,Y 336.441,Z 537.725,A -85,B 0,C 180,E1 -16246.504,E2 -16246.504} C_VEL
LIN {X 0,Y 340.754,Z 547.254,A -85,B 0,C 180,E1 -16247.45,E2 -16247.45} C_VEL
LIN {X 0,Y 334.905,Z 680.185,A -85,B 0,C 180,E1 -16250.255,E2 -16250.255} C_VEL
LIN {X 0,Y 333.591,Z 699.059,A -85,B 0,C 180,E1 -16250.752,E2 -16250.752} C_VEL
LIN {X 0,Y 331.955,Z 713.592,A -85,B 0,C 180,E1 -16251.303,E2 -16251.303} C_VEL
LIN {X 0,Y 330.089,Z 727.058,A -85,B 0,C 180,E1 -16251.978,E2 -16251.978} C_VEL
LIN {X 0,Y 328.16,Z 738.998,A -85,B 0,C 180,E1 -16252.721,E2 -16252.721} C_VEL
LIN {X 0,Y 325.875,Z 751.139,A -85,B 0,C 180,E1 -16253.625,E2 -16253.625} C_VEL
LIN {X 0,Y 323.465,Z 762.78,A -85,B 0,C 180,E1 -16254.657,E2 -16254.657} C_VEL
LIN {X 0,Y 320.427,Z 775.606,A -85,B 0,C 180,E1 -16255.994,E2 -16255.994} C_VEL
LIN {X 0,Y 317.77,Z 786.251,A -85,B 0,C 180,E1 -16257.298,E2 -16257.298} C_VEL
LIN {X 0,Y 315.024,Z 796.575,A -85,B 0,C 180,E1 -16258.756,E2 -16258.756} C_VEL
LIN {X 0,Y 312.25,Z 806.263,A -85,B 0,C 180,E1 -16260.32,E2 -16260.32} C_VEL
LIN {X 0,Y 309.371,Z 816.373,A -85,B 0,C 180,E1 -16262.222,E2 -16262.222} C_VEL
LIN {X 0,Y 306.847,Z 825.435,A -85,B 0,C 180,E1 -16264.204,E2 -16264.204} C_VEL
LIN {X 0,Y 304.484,Z 833.324,A -85,B 0,C 180,E1 -16266.177,E2 -16266.177} C_VEL
LIN {X 0,Y 302.355,Z 840.97,A -85,B 0,C 180,E1 -16268.398,E2 -16268.398} C_VEL
LIN {X 0,Y 300.488,Z 848.252,A -85,B 0,C 180,E1 -16270.887,E2 -16270.887} C_VEL
LIN {X 0,Y 299.244,Z 853.384,A -85,B 0,C 180,E1 -16272.928,E2 -16272.928} C_VEL
LIN {X 0,Y 298.045,Z 859.175,A -85,B 0,C 180,E1 -16275.681,E2 -16275.681} C_VEL
LIN {X 0,Y 297.34,Z 862.759,A -85,B 0,C 180,E1 -16277.718,E2 -16277.718} C_VEL
LIN {X 0,Y 296.752,Z 866.612,A -85,B 0,C 180,E1 -16280.458,E2 -16280.458} C_VEL
LIN {X 0,Y 296.573,Z 869.467,A -85,B 0,C 180,E1 -16283.195,E2 -16283.195} C_VEL
LIN {X 0,Y 296.499,Z 871.352,A -85,B 0,C 180,E1 -16285.922,E2 -16285.922} C_VEL
LIN {X 0,Y 296.518,Z 872.03,A -85,B 0,C 180,E1 -16287.283,E2 -16287.283} C_VEL
LIN {X 0,Y 296.473,Z 872.501,A -85,B 0,C 180,E1 -16290,E2 -16290} C_VEL
LIN {X 0,Y 296.518,Z 872.03,A -85,B 0,C 180,E1 -16292.717,E2 -16292.717} C_VEL
LIN {X 0,Y 296.511,Z 870.603,A -85,B 0,C 180,E1 -16295.44,E2 -16295.44} C_VEL
LIN {X 0,Y 296.622,Z 868.215,A -85,B 0,C 180,E1 -16298.173,E2 -16298.173} C_VEL
LIN {X 0,Y 297.138,Z 863.799,A -85,B 0,C 180,E1 -16301.598,E2 -16301.598} C_VEL
LIN {X 0,Y 297.747,Z 860.431,A -85,B 0,C 180,E1 -16303.653,E2 -16303.653} C_VEL
LIN {X 0,Y 298.879,Z 854.929,A -85,B 0,C 180,E1 -16306.39,E2 -16306.39} C_VEL
LIN {X 0,Y 300.058,Z 850.069,A -85,B 0,C 180,E1 -16308.433,E2 -16308.433} C_VEL
LIN {X 0,Y 301.936,Z 842.69,A -85,B 0,C 180,E1 -16311.049,E2 -16311.049} C_VEL
LIN {X 0,Y 303.805,Z 835.743,A -85,B 0,C 180,E1 -16313.157,E2 -16313.157} C_VEL
LIN {X 0,Y 305.977,Z 828.19,A -85,B 0,C 180,E1 -16315.145,E2 -16315.145} C_VEL
LIN {X 0,Y 308.464,Z 819.605,A -85,B 0,C 180,E1 -16317.108,E2 -16317.108} C_VEL
LIN {X 0,Y 311.244,Z 809.814,A -85,B 0,C 180,E1 -16319.043,E2 -16319.043} C_VEL
LIN {X 0,Y 314.127,Z 799.592,A -85,B 0,C 180,E1 -16320.782,E2 -16320.782} C_VEL
LIN {X 0,Y 316.725,Z 790.171,A -85,B 0,C 180,E1 -16322.177,E2 -16322.177} C_VEL
LIN {X 0,Y 319.757,Z 778.216,A -85,B 0,C 180,E1 -16323.708,E2 -16323.708} C_VEL
LIN {X 0,Y 322.396,Z 767.278,A -85,B 0,C 180,E1 -16324.905,E2 -16324.905} C_VEL
LIN {X 0,Y 324.794,Z 756.363,A -85,B 0,C 180,E1 -16325.939,E2 -16325.939} C_VEL
LIN {X 0,Y 327.341,Z 743.633,A -85,B 0,C 180,E1 -16326.952,E2 -16326.952} C_VEL
LIN {X 0,Y 329.546,Z 730.575,A -85,B 0,C 180,E1 -16327.82,E2 -16327.82} C_VEL
LIN {X 0,Y 331.497,Z 717.425,A -85,B 0,C 180,E1 -16328.518,E2 -16328.518} C_VEL
LIN {X 0,Y 333.108,Z 704.056,A -85,B 0,C 180,E1 -16329.072,E2 -16329.072} C_VEL
LIN {X 0,Y 334.275,Z 690.603,A -85,B 0,C 180,E1 -16329.493,E2 -16329.493} C_VEL
LIN {X 0,Y 335.97,Z 655.108,A -85,B 0,C 180,E1 -16330.278,E2 -16330.278} C_VEL
LIN {X 0,Y 339.69,Z 570.899,A -85,B 0,C 180,E1 -16332.053,E2 -16332.053} C_VEL
LIN {X 0,Y 340.676,Z 547.031,A -85,B 0,C 180,E1 -16332.568,E2 -16332.568} C_VEL
LIN {X 0,Y 333.198,Z 530.944,A -85,B 0,C 180,E1 -16334.222,E2 -16334.222} C_VEL
LIN {X 0,Y 326.718,Z 518.364,A -85,B 0,C 180,E1 -16335.716,E2 -16335.716} C_VEL
LIN {X 0,Y 319.219,Z 504.891,A -85,B 0,C 180,E1 -16337.539,E2 -16337.539} C_VEL
LIN {X 0,Y 313.202,Z 494.983,A -85,B 0,C 180,E1 -16339.085,E2 -16339.085} C_VEL
LIN {X 0,Y 309.639,Z 489.432,A -85,B 0,C 180,E1 -16340.041,E2 -16340.041} C_VEL
LIN {X 0,Y 306.558,Z 484.759,A -85,B 0,C 180,E1 -16340.897,E2 -16340.897} C_VEL
LIN {X 0,Y 302.905,Z 479.275,A -85,B 0,C 180,E1 -16341.953,E2 -16341.953} C_VEL
LIN {X 0,Y 299.754,Z 474.511,A -85,B 0,C 180,E1 -16342.959,E2 -16342.959} C_VEL
LIN {X 0,Y 298.473,Z 470.859,A -85,B 0,C 180,E1 -16344.562,E2 -16344.562} C_VEL
LIN {X 0,Y 298.404,Z 470.524,A -85,B 0,C 180,E1 -16345.171,E2 -16345.171} C_VEL
LIN {X 0,Y 298.394,Z 470.546,A -85,B 0,C 180,E1 -16348.791,E2 -16348.791} C_VEL
LIN {X 0,Y 298.448,Z 470.492,A -85,B 0,C 180,E1 -16351.903,E2 -16351.903} C_VEL
LIN {X 0,Y 298.476,Z 470.547,A -85,B 0,C 180,E1 -16354.923,E2 -16354.923} C_VEL
LIN {X 0,Y 298.428,Z 470.484,A -85,B 0,C 180,E1 -16359.314,E2 -16359.314} C_VEL
LIN {X 0,Y 298.528,Z 470.498,A -85,B 0,C 180,E1 -16362.179,E2 -16362.179} C_VEL
LIN {X 0,Y 298.587,Z 470.535,A -85,B 0,C 180,E1 -16364.994,E2 -16364.994} C_VEL
LIN {X 0,Y 298.585,Z 470.541,A -85,B 0,C 180,E1 -16369.146,E2 -16369.146} C_VEL
LIN {X 0,Y 298.735,Z 470.502,A -85,B 0,C 180,E1 -16371.885,E2 -16371.885} C_VEL
LIN {X 0,Y 298.652,Z 470.529,A -85,B 0,C 180,E1 -16374.599,E2 -16374.599} C_VEL
LIN {X 0,Y 298.917,Z 470.5,A -85,B 0,C 180,E1 -16378.652,E2 -16378.652} C_VEL
LIN {X 0,Y 298.917,Z 470.475,A -85,B 0,C 180,E1 -16381.347,E2 -16381.347} C_VEL
LIN {X 0,Y 298.786,Z 470.492,A -85,B 0,C 180,E1 -16386.754,E2 -16386.754} C_VEL
LIN {X 0,Y 298.674,Z 470.522,A -85,B 0,C 180,E1 -16389.48,E2 -16389.48} C_VEL
LIN {X 0,Y 298.545,Z 470.545,A -85,B 0,C 180,E1 -16393.615,E2 -16393.615} C_VEL
LIN {X 0,Y 298.542,Z 470.528,A -85,B 0,C 180,E1 -16396.409,E2 -16396.409} C_VEL
LIN {X 0,Y 298.491,Z 470.539,A -85,B 0,C 180,E1 -16399.647,E2 -16399.647} C_VEL
LIN {X 0,Y 298.422,Z 470.545,A -85,B 0,C 180,E1 -16403.6,E2 -16403.6} C_VEL
LIN {X 0,Y 298.478,Z 470.486,A -85,B 0,C 180,E1 -16406.575,E2 -16406.575} C_VEL
LIN {X 0,Y 298.415,Z 470.544,A -85,B 0,C 180,E1 -16409.641,E2 -16409.641} C_VEL
LIN {X 0,Y 298.389,Z 470.516,A -85,B 0,C 180,E1 -16412.8,E2 -16412.8} C_VEL
LIN {X 0,Y 298.479,Z 470.707,A -85,B 0,C 180,E1 -16416.695,E2 -16416.695} C_VEL
LIN {X 0,Y 298.653,Z 471.6,A -85,B 0,C 180,E1 -16417.062,E2 -16417.062} C_VEL
LIN {X 0,Y 300.092,Z 474.339,A -85,B 0,C 180,E1 -16417.586,E2 -16417.586} C_VEL
LIN {X 0,Y 302.526,Z 476.477,A -85,B 0,C 180,E1 -16418.293,E2 -16418.293} C_VEL
LIN {X 0,Y 304.581,Z 479.677,A -85,B 0,C 180,E1 -16418.959,E2 -16418.959} C_VEL
LIN {X 0,Y 307.138,Z 481.989,A -85,B 0,C 180,E1 -16419.737,E2 -16419.737} C_VEL
LIN {X 0,Y 309.716,Z 485.401,A -85,B 0,C 180,E1 -16420.593,E2 -16420.593} C_VEL
LIN {X 0,Y 312.363,Z 487.823,A -85,B 0,C 180,E1 -16421.457,E2 -16421.457} C_VEL
LIN {X 0,Y 315.37,Z 491.455,A -85,B 0,C 180,E1 -16422.52,E2 -16422.52} C_VEL
LIN {X 0,Y 318.103,Z 493.823,A -85,B 0,C 180,E1 -16423.491,E2 -16423.491} C_VEL
LIN {X 0,Y 321.261,Z 497.557,A -85,B 0,C 180,E1 -16424.712,E2 -16424.712} C_VEL
LIN {X 0,Y 323.865,Z 499.844,A -85,B 0,C 180,E1 -16425.734,E2 -16425.734} C_VEL
LIN {X 0,Y 326.851,Z 503.367,A -85,B 0,C 180,E1 -16426.976,E2 -16426.976} C_VEL
LIN {X 0,Y 329.552,Z 505.823,A -85,B 0,C 180,E1 -16428.088,E2 -16428.088} C_VEL
LIN {X 0,Y 332.971,Z 509.68,A -85,B 0,C 180,E1 -16429.559,E2 -16429.559} C_VEL
LIN {X 0,Y 335.45,Z 511.864,A -85,B 0,C 180,E1 -16430.623,E2 -16430.623} C_VEL
LIN {X 0,Y 338.648,Z 515.497,A -85,B 0,C 180,E1 -16432.056,E2 -16432.056} C_VEL
LIN {X 0,Y 341.584,Z 518.009,A -85,B 0,C 180,E1 -16433.36,E2 -16433.36} C_VEL
LIN {X 0,Y 344.922,Z 521.738,A -85,B 0,C 180,E1 -16434.935,E2 -16434.935} C_VEL
LIN {X 0,Y 348.163,Z 524.502,A -85,B 0,C 180,E1 -16436.466,E2 -16436.466} C_VEL
LIN {X 0,Y 351.26,Z 527.899,A -85,B 0,C 180,E1 -16438.021,E2 -16438.021} C_VEL
LIN {X 0,Y 354.786,Z 530.675,A -85,B 0,C 180,E1 -16439.791,E2 -16439.791} C_VEL
LIN {X 0,Y 357.848,Z 534.095,A -85,B 0,C 180,E1 -16441.479,E2 -16441.479} C_VEL
LIN {X 0,Y 361.626,Z 537.13,A -85,B 0,C 180,E1 -16443.609,E2 -16443.609} C_VEL
LIN {X 0,Y 364.812,Z 540.763,A -85,B 0,C 180,E1 -16445.581,E2 -16445.581} C_VEL
LIN {X 0,Y 368.057,Z 543.092,A -85,B 0,C 180,E1 -16447.672,E2 -16447.672} C_VEL
LIN {X 0,Y 369.18,Z 544.025,A -85,B 0,C 180,E1 -16448.42,E2 -16448.42} C_VEL
LIN {X 0,Y 371.715,Z 547.033,A -85,B 0,C 180,E1 -16450.349,E2 -16450.349} C_VEL
LIN {X 0,Y 374.738,Z 549.29,A -85,B 0,C 180,E1 -16452.737,E2 -16452.737} C_VEL
LIN {X 0,Y 376.69,Z 550.419,A -85,B 0,C 180,E1 -16454.448,E2 -16454.448} C_VEL
LIN {X 0,Y 378.625,Z 553.03,A -85,B 0,C 180,E1 -16456.488,E2 -16456.488} C_VEL
LIN {X 0,Y 380.726,Z 555,A -85,B 0,C 180,E1 -16459.039,E2 -16459.039} C_VEL
LIN {X 0,Y 382.475,Z 555.93,A -85,B 0,C 180,E1 -16461.547,E2 -16461.547} C_VEL
LIN {X 0,Y 383.909,Z 556.68,A -85,B 0,C 180,E1 -16464.395,E2 -16464.395} C_VEL
LIN {X 0,Y 384.685,Z 557.129,A -85,B 0,C 180,E1 -16466.858,E2 -16466.858} C_VEL
LIN {X 0,Y 384.987,Z 557.326,A -85,B 0,C 180,E1 -16468.954,E2 -16468.954} C_VEL
LIN {X 0,Y 384.987,Z 557.328,A -85,B 0,C 180,E1 -16471.046,E2 -16471.046} C_VEL
LIN {X 0,Y 384.685,Z 557.129,A -85,B 0,C 180,E1 -16473.142,E2 -16473.142} C_VEL
LIN {X 0,Y 383.912,Z 556.654,A -85,B 0,C 180,E1 -16475.604,E2 -16475.604} C_VEL
LIN {X 0,Y 382.472,Z 555.952,A -85,B 0,C 180,E1 -16478.453,E2 -16478.453} C_VEL
LIN {X 0,Y 380.737,Z 554.931,A -85,B 0,C 180,E1 -16480.96,E2 -16480.96} C_VEL
LIN {X 0,Y 378.752,Z 553.188,A -85,B 0,C 180,E1 -16483.353,E2 -16483.353} C_VEL
LIN {X 0,Y 376.69,Z 550.421,A -85,B 0,C 180,E1 -16485.55,E2 -16485.55} C_VEL
LIN {X 0,Y 373.531,Z 548.523,A -85,B 0,C 180,E1 -16488.232,E2 -16488.232} C_VEL
LIN {X 0,Y 370.539,Z 545.802,A -85,B 0,C 180,E1 -16490.552,E2 -16490.552} C_VEL
LIN {X 0,Y 368.5,Z 543.317,A -85,B 0,C 180,E1 -16492.047,E2 -16492.047} C_VEL
LIN {X 0,Y 365.145,Z 541.084,A -85,B 0,C 180,E1 -16494.202,E2 -16494.202} C_VEL
LIN {X 0,Y 361.96,Z 537.611,A -85,B 0,C 180,E1 -16496.19,E2 -16496.19} C_VEL
LIN {X 0,Y 360.88,Z 536.434,A -85,B 0,C 180,E1 -16496.832,E2 -16496.832} C_VEL
LIN {X 0,Y 357.326,Z 533.647,A -85,B 0,C 180,E1 -16498.81,E2 -16498.81} C_VEL
LIN {X 0,Y 354.026,Z 529.978,A -85,B 0,C 180,E1 -16500.594,E2 -16500.594} C_VEL
LIN {X 0,Y 350.532,Z 527.218,A -85,B 0,C 180,E1 -16502.342,E2 -16502.342} C_VEL
LIN {X 0,Y 347.336,Z 523.595,A -85,B 0,C 180,E1 -16503.944,E2 -16503.944} C_VEL
LIN {X 0,Y 343.519,Z 520.34,A -85,B 0,C 180,E1 -16505.738,E2 -16505.738} C_VEL
LIN {X 0,Y 340.798,Z 517.181,A -85,B 0,C 180,E1 -16507.009,E2 -16507.009} C_VEL
LIN {X 0,Y 337.097,Z 513.889,A -85,B 0,C 180,E1 -16508.648,E2 -16508.648} C_VEL
LIN {X 0,Y 334.606,Z 510.987,A -85,B 0,C 180,E1 -16509.748,E2 -16509.748} C_VEL
LIN {X 0,Y 330.837,Z 507.489,A -85,B 0,C 180,E1 -16511.349,E2 -16511.349} C_VEL
LIN {X 0,Y 328.876,Z 505.081,A -85,B 0,C 180,E1 -16512.19,E2 -16512.19} C_VEL
LIN {X 0,Y 325.322,Z 501.778,A -85,B 0,C 180,E1 -16513.649,E2 -16513.649} C_VEL
LIN {X 0,Y 323.025,Z 498.975,A -85,B 0,C 180,E1 -16514.611,E2 -16514.611} C_VEL
LIN {X 0,Y 319.624,Z 495.825,A -85,B 0,C 180,E1 -16515.918,E2 -16515.918} C_VEL
LIN {X 0,Y 317.44,Z 493.113,A -85,B 0,C 180,E1 -16516.754,E2 -16516.754} C_VEL
LIN {X 0,Y 314.25,Z 490.336,A -85,B 0,C 180,E1 -16517.862,E2 -16517.862} C_VEL
LIN {X 0,Y 311.725,Z 487.075,A -85,B 0,C 180,E1 -16518.758,E2 -16518.758} C_VEL
LIN {X 0,Y 308.493,Z 484.049,A -85,B 0,C 180,E1 -16519.804,E2 -16519.804} C_VEL
LIN {X 0,Y 306.7,Z 481.447,A -85,B 0,C 180,E1 -16520.408,E2 -16520.408} C_VEL
LIN {X 0,Y 304.012,Z 478.959,A -85,B 0,C 180,E1 -16521.222,E2 -16521.222} C_VEL
LIN {X 0,Y 302.013,Z 475.893,A -85,B 0,C 180,E1 -16521.86,E2 -16521.86} C_VEL
LIN {X 0,Y 299.774,Z 473.937,A -85,B 0,C 180,E1 -16522.509,E2 -16522.509} C_VEL
LIN {X 0,Y 298.552,Z 471.172,A -85,B 0,C 180,E1 -16523.054,E2 -16523.054} C_VEL
LIN {X 0,Y 298.483,Z 470.588,A -85,B 0,C 180,E1 -16523.559,E2 -16523.559} C_VEL
LIN {X 0,Y 298.389,Z 470.516,A -85,B 0,C 180,E1 -16527.2,E2 -16527.2} C_VEL
LIN {X 0,Y 298.425,Z 470.534,A -85,B 0,C 180,E1 -16530.615,E2 -16530.615} C_VEL
LIN {X 0,Y 298.47,Z 470.487,A -85,B 0,C 180,E1 -16533.477,E2 -16533.477} C_VEL
LIN {X 0,Y 298.424,Z 470.553,A -85,B 0,C 180,E1 -16536.699,E2 -16536.699} C_VEL
LIN {X 0,Y 298.518,Z 470.54,A -85,B 0,C 180,E1 -16540.756,E2 -16540.756} C_VEL
LIN {X 0,Y 298.586,Z 470.524,A -85,B 0,C 180,E1 -16544.995,E2 -16544.995} C_VEL
LIN {X 0,Y 298.586,Z 470.519,A -85,B 0,C 180,E1 -16549.147,E2 -16549.147} C_VEL
LIN {X 0,Y 298.748,Z 470.515,A -85,B 0,C 180,E1 -16551.886,E2 -16551.886} C_VEL
LIN {X 0,Y 298.653,Z 470.516,A -85,B 0,C 180,E1 -16554.599,E2 -16554.599} C_VEL
LIN {X 0,Y 298.917,Z 470.477,A -85,B 0,C 180,E1 -16558.653,E2 -16558.653} C_VEL
LIN {X 0,Y 298.917,Z 470.502,A -85,B 0,C 180,E1 -16561.348,E2 -16561.348} C_VEL
LIN {X 0,Y 298.782,Z 470.512,A -85,B 0,C 180,E1 -16566.754,E2 -16566.754} C_VEL
LIN {X 0,Y 298.731,Z 470.502,A -85,B 0,C 180,E1 -16567.905,E2 -16567.905} C_VEL
LIN {X 0,Y 298.048,Z 470.59,A -85,B 0,C 180,E1 -16569.029,E2 -16569.029} C_VEL
LIN {X 0,Y 295.093,Z 470.975,A -85,B 0,C 180,E1 -16570.855,E2 -16570.855} C_VEL
LIN {X 0,Y 292.606,Z 471.272,A -85,B 0,C 180,E1 -16572.338,E2 -16572.338} C_VEL
LIN {X 0,Y 291.575,Z 471.393,A -85,B 0,C 180,E1 -16573.489,E2 -16573.489} C_VEL
LIN {X 0,Y 291.511,Z 471.402,A -85,B 0,C 180,E1 -16573.879,E2 -16573.879} C_VEL
LIN {X 0,Y 291.48,Z 471.405,A -85,B 0,C 180,E1 -16576.818,E2 -16576.818} C_VEL
LIN {X 0,Y 291.446,Z 471.35,A -85,B 0,C 180,E1 -16579.875,E2 -16579.875} C_VEL
LIN {X 0,Y 291.411,Z 471.437,A -85,B 0,C 180,E1 -16584.204,E2 -16584.204} C_VEL
LIN {X 0,Y 291.412,Z 471.373,A -85,B 0,C 180,E1 -16587.273,E2 -16587.273} C_VEL
LIN {X 0,Y 291.334,Z 471.401,A -85,B 0,C 180,E1 -16590.437,E2 -16590.437} C_VEL
LIN {X 0,Y 291.349,Z 471.538,A -85,B 0,C 180,E1 -16593.833,E2 -16593.833} C_VEL
LIN {X 0,Y 292.153,Z 473.848,A -85,B 0,C 180,E1 -16594.971,E2 -16594.971} C_VEL
LIN {X 0,Y 295.254,Z 478.596,A -85,B 0,C 180,E1 -16596.095,E2 -16596.095} C_VEL
LIN {X 0,Y 297.118,Z 481.182,A -85,B 0,C 180,E1 -16596.683,E2 -16596.683} C_VEL
LIN {X 0,Y 301.193,Z 487.142,A -85,B 0,C 180,E1 -16597.93,E2 -16597.93} C_VEL
LIN {X 0,Y 308.065,Z 497.618,A -85,B 0,C 180,E1 -16599.903,E2 -16599.903} C_VEL
LIN {X 0,Y 314.444,Z 508.315,A -85,B 0,C 180,E1 -16601.623,E2 -16601.623} C_VEL
LIN {X 0,Y 321.764,Z 521.354,A -85,B 0,C 180,E1 -16603.474,E2 -16603.474} C_VEL
LIN {X 0,Y 329.159,Z 535.955,A -85,B 0,C 180,E1 -16605.245,E2 -16605.245} C_VEL
LIN {X 0,Y 335.401,Z 549.594,A -85,B 0,C 180,E1 -16606.679,E2 -16606.679} C_VEL
LIN {X 0,Y 330.034,Z 667.437,A -85,B 0,C 180,E1 -16609.196,E2 -16609.196} C_VEL
LIN {X 0,Y 328.655,Z 693.233,A -85,B 0,C 180,E1 -16609.795,E2 -16609.795} C_VEL
LIN {X 0,Y 326.648,Z 711.85,A -85,B 0,C 180,E1 -16610.453,E2 -16610.453} C_VEL
LIN {X 0,Y 324.736,Z 725.487,A -85,B 0,C 180,E1 -16611.126,E2 -16611.126} C_VEL
LIN {X 0,Y 322.448,Z 739.154,A -85,B 0,C 180,E1 -16611.98,E2 -16611.98} C_VEL
LIN {X 0,Y 320.154,Z 750.928,A -85,B 0,C 180,E1 -16612.867,E2 -16612.867} C_VEL
LIN {X 0,Y 317.656,Z 762.568,A -85,B 0,C 180,E1 -16613.91,E2 -16613.91} C_VEL
LIN {X 0,Y 314.507,Z 775.394,A -85,B 0,C 180,E1 -16615.263,E2 -16615.263} C_VEL
LIN {X 0,Y 312.083,Z 784.892,A -85,B 0,C 180,E1 -16616.432,E2 -16616.432} C_VEL
LIN {X 0,Y 308.876,Z 796.361,A -85,B 0,C 180,E1 -16618.062,E2 -16618.062} C_VEL
LIN {X 0,Y 306.007,Z 806.05,A -85,B 0,C 180,E1 -16619.652,E2 -16619.652} C_VEL
LIN {X 0,Y 303.426,Z 814.849,A -85,B 0,C 180,E1 -16621.313,E2 -16621.313} C_VEL
LIN {X 0,Y 300.39,Z 825.222,A -85,B 0,C 180,E1 -16623.608,E2 -16623.608} C_VEL
LIN {X 0,Y 297.9,Z 833.111,A -85,B 0,C 180,E1 -16625.616,E2 -16625.616} C_VEL
LIN {X 0,Y 295.843,Z 840.077,A -85,B 0,C 180,E1 -16627.661,E2 -16627.661} C_VEL
LIN {X 0,Y 294.183,Z 846.221,A -85,B 0,C 180,E1 -16629.733,E2 -16629.733} C_VEL
LIN {X 0,Y 292.341,Z 853.171,A -85,B 0,C 180,E1 -16632.512,E2 -16632.512} C_VEL
LIN {X 0,Y 291.235,Z 858.09,A -85,B 0,C 180,E1 -16634.855,E2 -16634.855} C_VEL
LIN {X 0,Y 290.337,Z 862.547,A -85,B 0,C 180,E1 -16637.417,E2 -16637.417} C_VEL
LIN {X 0,Y 289.683,Z 866.4,A -85,B 0,C 180,E1 -16640.222,E2 -16640.222} C_VEL
LIN {X 0,Y 289.475,Z 869.256,A -85,B 0,C 180,E1 -16643.028,E2 -16643.028} C_VEL
LIN {X 0,Y 289.412,Z 870.553,A -85,B 0,C 180,E1 -16644.641,E2 -16644.641} C_VEL
LIN {X 0,Y 289.422,Z 871.82,A -85,B 0,C 180,E1 -16647.216,E2 -16647.216} C_VEL
LIN {X 0,Y 289.393,Z 872.292,A -85,B 0,C 180,E1 -16650,E2 -16650} C_VEL
LIN {X 0,Y 289.422,Z 871.82,A -85,B 0,C 180,E1 -16652.784,E2 -16652.784} C_VEL
LIN {X 0,Y 289.433,Z 870.393,A -85,B 0,C 180,E1 -16655.574,E2 -16655.574} C_VEL
LIN {X 0,Y 289.544,Z 868.004,A -85,B 0,C 180,E1 -16658.374,E2 -16658.374} C_VEL
LIN {X 0,Y 290.119,Z 863.587,A -85,B 0,C 180,E1 -16661.882,E2 -16661.882} C_VEL
LIN {X 0,Y 290.773,Z 860.219,A -85,B 0,C 180,E1 -16663.987,E2 -16663.987} C_VEL
LIN {X 0,Y 291.974,Z 854.716,A -85,B 0,C 180,E1 -16666.789,E2 -16666.789} C_VEL
LIN {X 0,Y 293.23,Z 849.856,A -85,B 0,C 180,E1 -16668.878,E2 -16668.878} C_VEL
LIN {X 0,Y 295.125,Z 842.757,A -85,B 0,C 180,E1 -16671.461,E2 -16671.461} C_VEL
LIN {X 0,Y 297.165,Z 835.529,A -85,B 0,C 180,E1 -16673.706,E2 -16673.706} C_VEL
LIN {X 0,Y 299.479,Z 827.978,A -85,B 0,C 180,E1 -16675.73,E2 -16675.73} C_VEL
LIN {X 0,Y 302.057,Z 819.392,A -85,B 0,C 180,E1 -16677.732,E2 -16677.732} C_VEL
LIN {X 0,Y 304.96,Z 809.601,A -85,B 0,C 180,E1 -16679.701,E2 -16679.701} C_VEL
LIN {X 0,Y 307.974,Z 799.38,A -85,B 0,C 180,E1 -16681.466,E2 -16681.466} C_VEL
LIN {X 0,Y 310.68,Z 789.959,A -85,B 0,C 180,E1 -16682.881,E2 -16682.881} C_VEL
LIN {X 0,Y 313.815,Z 778.003,A -85,B 0,C 180,E1 -16684.435,E2 -16684.435} C_VEL
LIN {X 0,Y 316.531,Z 767.066,A -85,B 0,C 180,E1 -16685.649,E2 -16685.649} C_VEL
LIN {X 0,Y 319.399,Z 754.41,A -85,B 0,C 180,E1 -16686.841,E2 -16686.841} C_VEL
LIN {X 0,Y 321.918,Z 741.982,A -85,B 0,C 180,E1 -16687.82,E2 -16687.82} C_VEL
LIN {X 0,Y 324.073,Z 729.634,A -85,B 0,C 180,E1 -16688.634,E2 -16688.634} C_VEL
LIN {X 0,Y 325.961,Z 717.215,A -85,B 0,C 180,E1 -16689.297,E2 -16689.297} C_VEL
LIN {X 0,Y 327.621,Z 703.846,A -85,B 0,C 180,E1 -16689.855,E2 -16689.855} C_VEL
LIN {X 0,Y 328.82,Z 690.393,A -85,B 0,C 180,E1 -16690.281,E2 -16690.281} C_VEL
LIN {X 0,Y 330.657,Z 653.107,A -85,B 0,C 180,E1 -16691.113,E2 -16691.113} C_VEL
